LIN {X 0,Y 418.21,Z 141.387,A -85,B 0,C 180,E1 -10228.603,E2 -10228.603} C_VEL
LIN {X 0,Y 418.29,Z 141.379,A -85,B 0,C 180,E1 -10231.936,E2 -10231.936} C_VEL
LIN {X 0,Y 418.289,Z 141.382,A -85,B 0,C 180,E1 -10235.162,E2 -10235.162} C_VEL
LIN {X 0,Y 418.233,Z 141.384,A -85,B 0,C 180,E1 -10238.303,E2 -10238.303} C_VEL
LIN {X 0,Y 418.275,Z 141.384,A -85,B 0,C 180,E1 -10241.382,E2 -10241.382} C_VEL
LIN {X 0,Y 418.3,Z 141.376,A -85,B 0,C 180,E1 -10244.405,E2 -10244.405} C_VEL
LIN {X 0,Y 418.354,Z 141.373,A -85,B 0,C 180,E1 -10247.385,E2 -10247.385} C_VEL
LIN {X 0,Y 418.34,Z 141.371,A -85,B 0,C 180,E1 -10250.328,E2 -10250.328} C_VEL
LIN {X 0,Y 418.486,Z 141.357,A -85,B 0,C 180,E1 -10253.248,E2 -10253.248} C_VEL
LIN {X 0,Y 418.337,Z 141.375,A -85,B 0,C 180,E1 -10255.181,E2 -10255.181} C_VEL
LIN {X 0,Y 418.543,Z 141.346,A -85,B 0,C 180,E1 -10258.075,E2 -10258.075} C_VEL
LIN {X 0,Y 418.671,Z 141.33,A -85,B 0,C 180,E1 -10259.999,E2 -10259.999} C_VEL
LIN {X 0,Y 418.507,Z 141.356,A -85,B 0,C 180,E1 -10262.887,E2 -10262.887} C_VEL
LIN {X 0,Y 418.485,Z 141.36,A -85,B 0,C 180,E1 -10266.751,E2 -10266.751} C_VEL
LIN {X 0,Y 418.339,Z 141.371,A -85,B 0,C 180,E1 -10269.671,E2 -10269.671} C_VEL
LIN {X 0,Y 418.343,Z 141.373,A -85,B 0,C 180,E1 -10273,E2 -10273} C_VEL
LIN {X 0,Y 418.31,Z 141.379,A -85,B 0,C 180,E1 -10276.735,E2 -10276.735} C_VEL
LIN {X 0,Y 418.267,Z 141.381,A -85,B 0,C 180,E1 -10279.79,E2 -10279.79} C_VEL
LIN {X 0,Y 418.234,Z 141.387,A -85,B 0,C 180,E1 -10282.736,E2 -10282.736} C_VEL
LIN {X 0,Y 418.267,Z 141.382,A -85,B 0,C 180,E1 -10285.904,E2 -10285.904} C_VEL
LIN {X 0,Y 418.26,Z 141.381,A -85,B 0,C 180,E1 -10289.162,E2 -10289.162} C_VEL
LIN {X 0,Y 418.253,Z 141.382,A -85,B 0,C 180,E1 -10292.844,E2 -10292.844} C_VEL
LIN {X 0,Y 418.244,Z 141.388,A -85,B 0,C 180,E1 -10296.239,E2 -10296.239} C_VEL
LIN {X 0,Y 418.262,Z 141.384,A -85,B 0,C 180,E1 -10299.68,E2 -10299.68} C_VEL
LIN {X 0,Y 418.28,Z 141.381,A -85,B 0,C 180,E1 -10302.329,E2 -10302.329} C_VEL
LIN {X 0,Y 418.269,Z 141.38,A -85,B 0,C 180,E1 -10305.114,E2 -10305.114} C_VEL
LIN {X 0,Y 418.287,Z 141.383,A -85,B 0,C 180,E1 -10307.773,E2 -10307.773} C_VEL
LIN {X 0,Y 418.262,Z 141.385,A -85,B 0,C 180,E1 -10311.56,E2 -10311.56} C_VEL
LIN {X 0,Y 418.254,Z 141.383,A -85,B 0,C 180,E1 -10315.159,E2 -10315.159} C_VEL
LIN {X 0,Y 418.24,Z 141.388,A -85,B 0,C 180,E1 -10317.472,E2 -10317.472} C_VEL
LIN {X 0,Y 418.263,Z 141.381,A -85,B 0,C 180,E1 -10320.896,E2 -10320.896} C_VEL
LIN {X 0,Y 418.266,Z 141.381,A -85,B 0,C 180,E1 -10324.096,E2 -10324.096} C_VEL
LIN {X 0,Y 418.233,Z 141.389,A -85,B 0,C 180,E1 -10327.264,E2 -10327.264} C_VEL
LIN {X 0,Y 418.279,Z 141.378,A -85,B 0,C 180,E1 -10330.365,E2 -10330.365} C_VEL
LIN {X 0,Y 418.312,Z 141.381,A -85,B 0,C 180,E1 -10333.405,E2 -10333.405} C_VEL
LIN {X 0,Y 418.342,Z 141.374,A -85,B 0,C 180,E1 -10337,E2 -10337} C_VEL
LIN {X 0,Y 418.338,Z 141.371,A -85,B 0,C 180,E1 -10340.329,E2 -10340.329} C_VEL
LIN {X 0,Y 418.491,Z 141.358,A -85,B 0,C 180,E1 -10343.249,E2 -10343.249} C_VEL
LIN {X 0,Y 418.338,Z 141.377,A -85,B 0,C 180,E1 -10345.182,E2 -10345.182} C_VEL
LIN {X 0,Y 418.541,Z 141.346,A -85,B 0,C 180,E1 -10348.076,E2 -10348.076} C_VEL
LIN {X 0,Y 418.669,Z 141.33,A -85,B 0,C 180,E1 -10350.001,E2 -10350.001} C_VEL
LIN {X 0,Y 418.507,Z 141.357,A -85,B 0,C 180,E1 -10352.888,E2 -10352.888} C_VEL
LIN {X 0,Y 418.492,Z 141.358,A -85,B 0,C 180,E1 -10356.752,E2 -10356.752} C_VEL
LIN {X 0,Y 418.339,Z 141.371,A -85,B 0,C 180,E1 -10359.672,E2 -10359.672} C_VEL
LIN {X 0,Y 418.32,Z 141.377,A -85,B 0,C 180,E1 -10363.332,E2 -10363.332} C_VEL
LIN {X 0,Y 417.618,Z 141.465,A -85,B 0,C 180,E1 -10363.869,E2 -10363.869} C_VEL
LIN {X 0,Y 411.929,Z 142.175,A -85,B 0,C 180,E1 -10365.56,E2 -10365.56} C_VEL
LIN {X 0,Y 411.331,Z 142.25,A -85,B 0,C 180,E1 -10366.109,E2 -10366.109} C_VEL
LIN {X 0,Y 411.337,Z 142.3,A -85,B 0,C 180,E1 -10366.375,E2 -10366.375} C_VEL
LIN {X 0,Y 412.888,Z 151.501,A -85,B 0,C 180,E1 -10368.612,E2 -10368.612} C_VEL
LIN {X 0,Y 412.993,Z 152.785,A -85,B 0,C 180,E1 -10368.865,E2 -10368.865} C_VEL
LIN {X 0,Y 417.017,Z 172.236,A -85,B 0,C 180,E1 -10369.411,E2 -10369.411} C_VEL
LIN {X 0,Y 415.681,Z 260.265,A -85,B 0,C 180,E1 -10371.012,E2 -10371.012} C_VEL
LIN {X 0,Y 415.299,Z 273.928,A -85,B 0,C 180,E1 -10371.47,E2 -10371.47} C_VEL
LIN {X 0,Y 414.856,Z 286.236,A -85,B 0,C 180,E1 -10372.079,E2 -10372.079} C_VEL
LIN {X 0,Y 414.377,Z 297.489,A -85,B 0,C 180,E1 -10372.829,E2 -10372.829} C_VEL
LIN {X 0,Y 413.625,Z 308.356,A -85,B 0,C 180,E1 -10373.743,E2 -10373.743} C_VEL
LIN {X 0,Y 412.896,Z 319.455,A -85,B 0,C 180,E1 -10374.916,E2 -10374.916} C_VEL
LIN {X 0,Y 412.3,Z 328.343,A -85,B 0,C 180,E1 -10376.083,E2 -10376.083} C_VEL
LIN {X 0,Y 411.685,Z 336.809,A -85,B 0,C 180,E1 -10377.448,E2 -10377.448} C_VEL
LIN {X 0,Y 411.157,Z 344.341,A -85,B 0,C 180,E1 -10378.949,E2 -10378.949} C_VEL
LIN {X 0,Y 410.667,Z 350.919,A -85,B 0,C 180,E1 -10380.607,E2 -10380.607} C_VEL
LIN {X 0,Y 410.404,Z 355.393,A -85,B 0,C 180,E1 -10382.064,E2 -10382.064} C_VEL
LIN {X 0,Y 410.11,Z 359.41,A -85,B 0,C 180,E1 -10383.846,E2 -10383.846} C_VEL
LIN {X 0,Y 409.895,Z 362.062,A -85,B 0,C 180,E1 -10385.66,E2 -10385.66} C_VEL
LIN {X 0,Y 409.854,Z 363.037,A -85,B 0,C 180,E1 -10386.883,E2 -10386.883} C_VEL
LIN {X 0,Y 409.846,Z 363.428,A -85,B 0,C 180,E1 -10388.122,E2 -10388.122} C_VEL
LIN {X 0,Y 409.88,Z 363.07,A -85,B 0,C 180,E1 -10389.504,E2 -10389.504} C_VEL
LIN {X 0,Y 410.015,Z 361.754,A -85,B 0,C 180,E1 -10391.046,E2 -10391.046} C_VEL
LIN {X 0,Y 410.216,Z 359.494,A -85,B 0,C 180,E1 -10392.55,E2 -10392.55} C_VEL
LIN {X 0,Y 410.428,Z 356.324,A -85,B 0,C 180,E1 -10394.013,E2 -10394.013} C_VEL
LIN {X 0,Y 410.724,Z 352.199,A -85,B 0,C 180,E1 -10395.449,E2 -10395.449} C_VEL
LIN {X 0,Y 411.192,Z 347,A -85,B 0,C 180,E1 -10396.87,E2 -10396.87} C_VEL
LIN {X 0,Y 411.676,Z 340.719,A -85,B 0,C 180,E1 -10398.258,E2 -10398.258} C_VEL
LIN {X 0,Y 412.308,Z 333.087,A -85,B 0,C 180,E1 -10399.63,E2 -10399.63} C_VEL
LIN {X 0,Y 413.033,Z 323.793,A -85,B 0,C 180,E1 -10400.982,E2 -10400.982} C_VEL
LIN {X 0,Y 413.785,Z 313.743,A -85,B 0,C 180,E1 -10402.158,E2 -10402.158} C_VEL
LIN {X 0,Y 414.575,Z 303.217,A -85,B 0,C 180,E1 -10403.149,E2 -10403.149} C_VEL
LIN {X 0,Y 415.31,Z 291.58,A -85,B 0,C 180,E1 -10404.015,E2 -10404.015} C_VEL
LIN {X 0,Y 415.854,Z 279.546,A -85,B 0,C 180,E1 -10404.694,E2 -10404.694} C_VEL
LIN {X 0,Y 416.243,Z 267.043,A -85,B 0,C 180,E1 -10405.202,E2 -10405.202} C_VEL
LIN {X 0,Y 416.569,Z 254.522,A -85,B 0,C 180,E1 -10405.52,E2 -10405.52} C_VEL
LIN {X 0,Y 417.79,Z 172.296,A -85,B 0,C 180,E1 -10407.018,E2 -10407.018} C_VEL
LIN {X 0,Y 413.907,Z 155.246,A -85,B 0,C 180,E1 -10407.558,E2 -10407.558} C_VEL
LIN {X 0,Y 413.389,Z 153.267,A -85,B 0,C 180,E1 -10407.657,E2 -10407.657} C_VEL
LIN {X 0,Y 411.253,Z 142.258,A -85,B 0,C 180,E1 -10410.349,E2 -10410.349} C_VEL
LIN {X 0,Y 411.236,Z 142.264,A -85,B 0,C 180,E1 -10413.62,E2 -10413.62} C_VEL
LIN {X 0,Y 411.198,Z 142.27,A -85,B 0,C 180,E1 -10416.853,E2 -10416.853} C_VEL
LIN {X 0,Y 411.218,Z 142.262,A -85,B 0,C 180,E1 -10420.051,E2 -10420.051} C_VEL
LIN {X 0,Y 411.267,Z 142.259,A -85,B 0,C 180,E1 -10423.132,E2 -10423.132} C_VEL
LIN {X 0,Y 411.31,Z 142.253,A -85,B 0,C 180,E1 -10426.897,E2 -10426.897} C_VEL
LIN {X 0,Y 411.294,Z 142.252,A -85,B 0,C 180,E1 -10430.162,E2 -10430.162} C_VEL
LIN {X 0,Y 411.395,Z 142.24,A -85,B 0,C 180,E1 -10433.133,E2 -10433.133} C_VEL
LIN {X 0,Y 411.295,Z 142.25,A -85,B 0,C 180,E1 -10435.099,E2 -10435.099} C_VEL
LIN {X 0,Y 411.507,Z 142.229,A -85,B 0,C 180,E1 -10438.043,E2 -10438.043} C_VEL
LIN {X 0,Y 411.385,Z 142.239,A -85,B 0,C 180,E1 -10440.979,E2 -10440.979} C_VEL
LIN {X 0,Y 411.431,Z 142.227,A -85,B 0,C 180,E1 -10442.938,E2 -10442.938} C_VEL
LIN {X 0,Y 411.432,Z 142.235,A -85,B 0,C 180,E1 -10445.883,E2 -10445.883} C_VEL
LIN {X 0,Y 411.31,Z 142.247,A -85,B 0,C 180,E1 -10448.847,E2 -10448.847} C_VEL
LIN {X 0,Y 411.273,Z 142.251,A -85,B 0,C 180,E1 -10451.834,E2 -10451.834} C_VEL
LIN {X 0,Y 411.211,Z 142.255,A -85,B 0,C 180,E1 -10454.855,E2 -10454.855} C_VEL
LIN {X 0,Y 411.161,Z 142.267,A -85,B 0,C 180,E1 -10457.92,E2 -10457.92} C_VEL
LIN {X 0,Y 411.182,Z 142.264,A -85,B 0,C 180,E1 -10461.035,E2 -10461.035} C_VEL
LIN {X 0,Y 411.176,Z 142.262,A -85,B 0,C 180,E1 -10464.219,E2 -10464.219} C_VEL
LIN {X 0,Y 411.145,Z 142.266,A -85,B 0,C 180,E1 -10467.486,E2 -10467.486} C_VEL
LIN {X 0,Y 411.197,Z 142.263,A -85,B 0,C 180,E1 -10469.714,E2 -10469.714} C_VEL
LIN {X 0,Y 411.209,Z 142.266,A -85,B 0,C 180,E1 -10473.156,E2 -10473.156} C_VEL
LIN {X 0,Y 411.197,Z 142.264,A -85,B 0,C 180,E1 -10476.552,E2 -10476.552} C_VEL
LIN {X 0,Y 411.174,Z 142.266,A -85,B 0,C 180,E1 -10479.72,E2 -10479.72} C_VEL
LIN {X 0,Y 411.167,Z 142.268,A -85,B 0,C 180,E1 -10483.135,E2 -10483.135} C_VEL
LIN {X 0,Y 411.17,Z 142.269,A -85,B 0,C 180,E1 -10485.881,E2 -10485.881} C_VEL
LIN {X 0,Y 411.156,Z 142.272,A -85,B 0,C 180,E1 -10488.774,E2 -10488.774} C_VEL
LIN {X 0,Y 411.191,Z 142.268,A -85,B 0,C 180,E1 -10492.025,E2 -10492.025} C_VEL
LIN {X 0,Y 411.211,Z 142.264,A -85,B 0,C 180,E1 -10495.666,E2 -10495.666} C_VEL
LIN {X 0,Y 411.194,Z 142.267,A -85,B 0,C 180,E1 -10499.152,E2 -10499.152} C_VEL
LIN {X 0,Y 411.26,Z 142.396,A -85,B 0,C 180,E1 -10501.489,E2 -10501.489} C_VEL
LIN {X 0,Y 413.905,Z 154.634,A -85,B 0,C 180,E1 -10504.149,E2 -10504.149} C_VEL
LIN {X 0,Y 414.568,Z 159.685,A -85,B 0,C 180,E1 -10505.191,E2 -10505.191} C_VEL
LIN {X 0,Y 413.326,Z 177.24,A -85,B 0,C 180,E1 -10508.556,E2 -10508.556} C_VEL
LIN {X 0,Y 412.781,Z 186.857,A -85,B 0,C 180,E1 -10510.376,E2 -10510.376} C_VEL
LIN {X 0,Y 416.686,Z 211.598,A -85,B 0,C 180,E1 -10511.057,E2 -10511.057} C_VEL
LIN {X 0,Y 417.247,Z 218.282,A -85,B 0,C 180,E1 -10511.212,E2 -10511.212} C_VEL
LIN {X 0,Y 416.163,Z 296.183,A -85,B 0,C 180,E1 -10512.652,E2 -10512.652} C_VEL
LIN {X 0,Y 415.507,Z 309.921,A -85,B 0,C 180,E1 -10513.099,E2 -10513.099} C_VEL
LIN {X 0,Y 414.819,Z 322.351,A -85,B 0,C 180,E1 -10513.703,E2 -10513.703} C_VEL
LIN {X 0,Y 414.049,Z 334.29,A -85,B 0,C 180,E1 -10514.493,E2 -10514.493} C_VEL
LIN {X 0,Y 413.192,Z 346.036,A -85,B 0,C 180,E1 -10515.495,E2 -10515.495} C_VEL
LIN {X 0,Y 412.425,Z 356.164,A -85,B 0,C 180,E1 -10516.574,E2 -10516.574} C_VEL
LIN {X 0,Y 411.663,Z 366.341,A -85,B 0,C 180,E1 -10517.928,E2 -10517.928} C_VEL
LIN {X 0,Y 410.915,Z 375.306,A -85,B 0,C 180,E1 -10519.405,E2 -10519.405} C_VEL
LIN {X 0,Y 410.462,Z 382.511,A -85,B 0,C 180,E1 -10520.887,E2 -10520.887} C_VEL
LIN {X 0,Y 410.174,Z 389.097,A -85,B 0,C 180,E1 -10522.616,E2 -10522.616} C_VEL
LIN {X 0,Y 409.99,Z 393.452,A -85,B 0,C 180,E1 -10524.096,E2 -10524.096} C_VEL
LIN {X 0,Y 410.009,Z 395.771,A -85,B 0,C 180,E1 -10525.083,E2 -10525.083} C_VEL
LIN {X 0,Y 409.941,Z 397.615,A -85,B 0,C 180,E1 -10526.067,E2 -10526.067} C_VEL
LIN {X 0,Y 409.973,Z 399.015,A -85,B 0,C 180,E1 -10527.052,E2 -10527.052} C_VEL
LIN {X 0,Y 410.02,Z 400.015,A -85,B 0,C 180,E1 -10528.035,E2 -10528.035} C_VEL
LIN {X 0,Y 409.983,Z 400.617,A -85,B 0,C 180,E1 -10529.017,E2 -10529.017} C_VEL
LIN {X 0,Y 409.979,Z 400.785,A -85,B 0,C 180,E1 -10529.999,E2 -10529.999} C_VEL
LIN {X 0,Y 409.983,Z 400.538,A -85,B 0,C 180,E1 -10530.982,E2 -10530.982} C_VEL
LIN {X 0,Y 410.02,Z 399.899,A -85,B 0,C 180,E1 -10531.964,E2 -10531.964} C_VEL
LIN {X 0,Y 409.976,Z 398.86,A -85,B 0,C 180,E1 -10532.947,E2 -10532.947} C_VEL
LIN {X 0,Y 409.943,Z 397.366,A -85,B 0,C 180,E1 -10533.932,E2 -10533.932} C_VEL
LIN {X 0,Y 410.002,Z 394.315,A -85,B 0,C 180,E1 -10535.409,E2 -10535.409} C_VEL
LIN {X 0,Y 410.095,Z 390.185,A -85,B 0,C 180,E1 -10536.889,E2 -10536.889} C_VEL
LIN {X 0,Y 410.373,Z 383.845,A -85,B 0,C 180,E1 -10538.618,E2 -10538.618} C_VEL
LIN {X 0,Y 410.733,Z 376.931,A -85,B 0,C 180,E1 -10540.101,E2 -10540.101} C_VEL
LIN {X 0,Y 411.244,Z 369.875,A -85,B 0,C 180,E1 -10541.334,E2 -10541.334} C_VEL
LIN {X 0,Y 411.812,Z 361.367,A -85,B 0,C 180,E1 -10542.567,E2 -10542.567} C_VEL
LIN {X 0,Y 412.504,Z 350.848,A -85,B 0,C 180,E1 -10543.799,E2 -10543.799} C_VEL
LIN {X 0,Y 413.334,Z 339.017,A -85,B 0,C 180,E1 -10544.902,E2 -10544.902} C_VEL
LIN {X 0,Y 414.107,Z 327.155,A -85,B 0,C 180,E1 -10545.756,E2 -10545.756} C_VEL
LIN {X 0,Y 414.793,Z 314.852,A -85,B 0,C 180,E1 -10546.423,E2 -10546.423} C_VEL
LIN {X 0,Y 415.336,Z 302.328,A -85,B 0,C 180,E1 -10546.907,E2 -10546.907} C_VEL
LIN {X 0,Y 415.652,Z 287.89,A -85,B 0,C 180,E1 -10547.242,E2 -10547.242} C_VEL
LIN {X 0,Y 416.483,Z 215.312,A -85,B 0,C 180,E1 -10548.55,E2 -10548.55} C_VEL
LIN {X 0,Y 412.522,Z 188.027,A -85,B 0,C 180,E1 -10549.241,E2 -10549.241} C_VEL
LIN {X 0,Y 413.776,Z 168.398,A -85,B 0,C 180,E1 -10552.995,E2 -10552.995} C_VEL
LIN {X 0,Y 414.447,Z 158.976,A -85,B 0,C 180,E1 -10554.815,E2 -10554.815} C_VEL
LIN {X 0,Y 413.035,Z 150.76,A -85,B 0,C 180,E1 -10556.529,E2 -10556.529} C_VEL
LIN {X 0,Y 411.316,Z 142.251,A -85,B 0,C 180,E1 -10558.373,E2 -10558.373} C_VEL
LIN {X 0,Y 411.167,Z 142.271,A -85,B 0,C 180,E1 -10561.997,E2 -10561.997} C_VEL
LIN {X 0,Y 411.211,Z 142.259,A -85,B 0,C 180,E1 -10564.878,E2 -10564.878} C_VEL
LIN {X 0,Y 411.208,Z 142.263,A -85,B 0,C 180,E1 -10568.168,E2 -10568.168} C_VEL
LIN {X 0,Y 411.165,Z 142.266,A -85,B 0,C 180,E1 -10571.228,E2 -10571.228} C_VEL
LIN {X 0,Y 411.176,Z 142.264,A -85,B 0,C 180,E1 -10574.49,E2 -10574.49} C_VEL
LIN {X 0,Y 411.177,Z 142.265,A -85,B 0,C 180,E1 -10578.194,E2 -10578.194} C_VEL
LIN {X 0,Y 411.21,Z 142.259,A -85,B 0,C 180,E1 -10580.774,E2 -10580.774} C_VEL
LIN {X 0,Y 411.196,Z 142.261,A -85,B 0,C 180,E1 -10584.471,E2 -10584.471} C_VEL
LIN {X 0,Y 411.206,Z 142.26,A -85,B 0,C 180,E1 -10586.873,E2 -10586.873} C_VEL
LIN {X 0,Y 411.232,Z 142.256,A -85,B 0,C 180,E1 -10590.644,E2 -10590.644} C_VEL
LIN {X 0,Y 411.237,Z 142.26,A -85,B 0,C 180,E1 -10593.619,E2 -10593.619} C_VEL
LIN {X 0,Y 411.202,Z 142.262,A -85,B 0,C 180,E1 -10596.852,E2 -10596.852} C_VEL
LIN {X 0,Y 411.213,Z 142.259,A -85,B 0,C 180,E1 -10600.05,E2 -10600.05} C_VEL
LIN {X 0,Y 411.261,Z 142.259,A -85,B 0,C 180,E1 -10603.131,E2 -10603.131} C_VEL
LIN {X 0,Y 411.304,Z 142.252,A -85,B 0,C 180,E1 -10606.895,E2 -10606.895} C_VEL
LIN {X 0,Y 411.292,Z 142.249,A -85,B 0,C 180,E1 -10610.161,E2 -10610.161} C_VEL
LIN {X 0,Y 411.45,Z 142.234,A -85,B 0,C 180,E1 -10613.132,E2 -10613.132} C_VEL
LIN {X 0,Y 411.308,Z 142.252,A -85,B 0,C 180,E1 -10615.098,E2 -10615.098} C_VEL
LIN {X 0,Y 411.512,Z 142.221,A -85,B 0,C 180,E1 -10618.042,E2 -10618.042} C_VEL
LIN {X 0,Y 411.64,Z 142.205,A -85,B 0,C 180,E1 -10619.999,E2 -10619.999} C_VEL
LIN {X 0,Y 411.463,Z 142.233,A -85,B 0,C 180,E1 -10622.937,E2 -10622.937} C_VEL
LIN {X 0,Y 411.449,Z 142.234,A -85,B 0,C 180,E1 -10626.867,E2 -10626.867} C_VEL
LIN {X 0,Y 411.291,Z 142.249,A -85,B 0,C 180,E1 -10629.838,E2 -10629.838} C_VEL
LIN {X 0,Y 411.302,Z 142.249,A -85,B 0,C 180,E1 -10633.104,E2 -10633.104} C_VEL
LIN {X 0,Y 411.259,Z 142.256,A -85,B 0,C 180,E1 -10636.868,E2 -10636.868} C_VEL
LIN {X 0,Y 411.227,Z 142.259,A -85,B 0,C 180,E1 -10639.986,E2 -10639.986} C_VEL
LIN {X 0,Y 411.199,Z 142.261,A -85,B 0,C 180,E1 -10643.147,E2 -10643.147} C_VEL
LIN {X 0,Y 411.234,Z 142.262,A -85,B 0,C 180,E1 -10646.38,E2 -10646.38} C_VEL
LIN {X 0,Y 411.196,Z 142.262,A -85,B 0,C 180,E1 -10649.712,E2 -10649.712} C_VEL
LIN {X 0,Y 411.202,Z 142.26,A -85,B 0,C 180,E1 -10653.155,E2 -10653.155} C_VEL
LIN {X 0,Y 411.191,Z 142.263,A -85,B 0,C 180,E1 -10656.553,E2 -10656.553} C_VEL
LIN {X 0,Y 411.224,Z 142.261,A -85,B 0,C 180,E1 -10659.73,E2 -10659.73} C_VEL
LIN {X 0,Y 411.226,Z 142.257,A -85,B 0,C 180,E1 -10663.126,E2 -10663.126} C_VEL
LIN {X 0,Y 411.235,Z 142.263,A -85,B 0,C 180,E1 -10665.871,E2 -10665.871} C_VEL
LIN {X 0,Y 411.205,Z 142.26,A -85,B 0,C 180,E1 -10668.764,E2 -10668.764} C_VEL
LIN {X 0,Y 411.2,Z 142.264,A -85,B 0,C 180,E1 -10672.028,E2 -10672.028} C_VEL
LIN {X 0,Y 411.201,Z 142.267,A -85,B 0,C 180,E1 -10675.667,E2 -10675.667} C_VEL
LIN {X 0,Y 411.184,Z 142.264,A -85,B 0,C 180,E1 -10679.153,E2 -10679.153} C_VEL
LIN {X 0,Y 411.254,Z 142.253,A -85,B 0,C 180,E1 -10682.523,E2 -10682.523} C_VEL
LIN {X 0,Y 411.222,Z 142.261,A -85,B 0,C 180,E1 -10685.785,E2 -10685.785} C_VEL
LIN {X 0,Y 411.192,Z 142.263,A -85,B 0,C 180,E1 -10688.966,E2 -10688.966} C_VEL
LIN {X 0,Y 411.248,Z 142.255,A -85,B 0,C 180,E1 -10692.085,E2 -10692.085} C_VEL
LIN {X 0,Y 411.256,Z 142.258,A -85,B 0,C 180,E1 -10695.148,E2 -10695.148} C_VEL
LIN {X 0,Y 411.28,Z 142.25,A -85,B 0,C 180,E1 -10698.168,E2 -10698.168} C_VEL
LIN {X 0,Y 411.478,Z 142.225,A -85,B 0,C 180,E1 -10702.147,E2 -10702.147} C_VEL
LIN {X 0,Y 411.473,Z 142.226,A -85,B 0,C 180,E1 -10704.119,E2 -10704.119} C_VEL
LIN {X 0,Y 411.51,Z 142.221,A -85,B 0,C 180,E1 -10708.043,E2 -10708.043} C_VEL
LIN {X 0,Y 411.639,Z 142.205,A -85,B 0,C 180,E1 -10710.001,E2 -10710.001} C_VEL
LIN {X 0,Y 411.463,Z 142.235,A -85,B 0,C 180,E1 -10712.938,E2 -10712.938} C_VEL
LIN {X 0,Y 411.458,Z 142.235,A -85,B 0,C 180,E1 -10716.868,E2 -10716.868} C_VEL
LIN {X 0,Y 411.291,Z 142.249,A -85,B 0,C 180,E1 -10719.839,E2 -10719.839} C_VEL
LIN {X 0,Y 411.284,Z 142.253,A -85,B 0,C 180,E1 -10723.32,E2 -10723.32} C_VEL
LIN {X 0,Y 411.331,Z 142.25,A -85,B 0,C 180,E1 -10726.109,E2 -10726.109} C_VEL
LIN {X 0,Y 411.267,Z 142.94,A -85,B 0,C 180,E1 -10726.499,E2 -10726.499} C_VEL
LIN {X 0,Y 410.694,Z 145.504,A -85,B 0,C 180,E1 -10727.091,E2 -10727.091} C_VEL
LIN {X 0,Y 409.217,Z 149.691,A -85,B 0,C 180,E1 -10727.933,E2 -10727.933} C_VEL
LIN {X 0,Y 408.351,Z 154.177,A -85,B 0,C 180,E1 -10728.364,E2 -10728.364} C_VEL
LIN {X 0,Y 407.985,Z 159.599,A -85,B 0,C 180,E1 -10728.712,E2 -10728.712} C_VEL
LIN {X 0,Y 408.345,Z 163.41,A -85,B 0,C 180,E1 -10728.858,E2 -10728.858} C_VEL
LIN {X 0,Y 410.228,Z 173.002,A -85,B 0,C 180,E1 -10729.125,E2 -10729.125} C_VEL
LIN {X 0,Y 408.875,Z 259.99,A -85,B 0,C 180,E1 -10730.731,E2 -10730.731} C_VEL
LIN {X 0,Y 408.466,Z 273.511,A -85,B 0,C 180,E1 -10731.182,E2 -10731.182} C_VEL
LIN {X 0,Y 408.031,Z 285.861,A -85,B 0,C 180,E1 -10731.793,E2 -10731.793} C_VEL
LIN {X 0,Y 407.518,Z 297.436,A -85,B 0,C 180,E1 -10732.565,E2 -10732.565} C_VEL
LIN {X 0,Y 406.701,Z 308.993,A -85,B 0,C 180,E1 -10733.553,E2 -10733.553} C_VEL
LIN {X 0,Y 405.986,Z 319.521,A -85,B 0,C 180,E1 -10734.685,E2 -10734.685} C_VEL
LIN {X 0,Y 405.298,Z 329.093,A -85,B 0,C 180,E1 -10735.967,E2 -10735.967} C_VEL
LIN {X 0,Y 404.63,Z 337.874,A -85,B 0,C 180,E1 -10737.425,E2 -10737.425} C_VEL
LIN {X 0,Y 404.131,Z 344.84,A -85,B 0,C 180,E1 -10738.855,E2 -10738.855} C_VEL
LIN {X 0,Y 403.678,Z 350.622,A -85,B 0,C 180,E1 -10740.325,E2 -10740.325} C_VEL
LIN {X 0,Y 403.301,Z 356.025,A -85,B 0,C 180,E1 -10742.107,E2 -10742.107} C_VEL
LIN {X 0,Y 403.026,Z 359.958,A -85,B 0,C 180,E1 -10743.92,E2 -10743.92} C_VEL
LIN {X 0,Y 402.853,Z 361.822,A -85,B 0,C 180,E1 -10745.15,E2 -10745.15} C_VEL
LIN {X 0,Y 402.769,Z 363.225,A -85,B 0,C 180,E1 -10746.616,E2 -10746.616} C_VEL
LIN {X 0,Y 402.765,Z 363.752,A -85,B 0,C 180,E1 -10748.26,E2 -10748.26} C_VEL
LIN {X 0,Y 402.823,Z 362.965,A -85,B 0,C 180,E1 -10750.207,E2 -10750.207} C_VEL
LIN {X 0,Y 403.078,Z 360.668,A -85,B 0,C 180,E1 -10752.167,E2 -10752.167} C_VEL
LIN {X 0,Y 403.275,Z 358.103,A -85,B 0,C 180,E1 -10753.52,E2 -10753.52} C_VEL
LIN {X 0,Y 403.548,Z 354.525,A -85,B 0,C 180,E1 -10754.942,E2 -10754.942} C_VEL
LIN {X 0,Y 404.033,Z 348.955,A -85,B 0,C 180,E1 -10756.638,E2 -10756.638} C_VEL
LIN {X 0,Y 404.651,Z 341.748,A -85,B 0,C 180,E1 -10758.317,E2 -10758.317} C_VEL
LIN {X 0,Y 405.322,Z 334.19,A -85,B 0,C 180,E1 -10759.724,E2 -10759.724} C_VEL
LIN {X 0,Y 406.102,Z 324.741,A -85,B 0,C 180,E1 -10761.149,E2 -10761.149} C_VEL
LIN {X 0,Y 406.911,Z 314.507,A -85,B 0,C 180,E1 -10762.378,E2 -10762.378} C_VEL
LIN {X 0,Y 407.841,Z 302.963,A -85,B 0,C 180,E1 -10763.481,E2 -10763.481} C_VEL
LIN {X 0,Y 408.525,Z 292.263,A -85,B 0,C 180,E1 -10764.287,E2 -10764.287} C_VEL
LIN {X 0,Y 409.116,Z 279.829,A -85,B 0,C 180,E1 -10765.002,E2 -10765.002} C_VEL
LIN {X 0,Y 409.587,Z 266.535,A -85,B 0,C 180,E1 -10765.543,E2 -10765.543} C_VEL
LIN {X 0,Y 409.9,Z 252.754,A -85,B 0,C 180,E1 -10765.877,E2 -10765.877} C_VEL
LIN {X 0,Y 411.101,Z 173.169,A -85,B 0,C 180,E1 -10767.36,E2 -10767.36} C_VEL
LIN {X 0,Y 407.478,Z 157.271,A -85,B 0,C 180,E1 -10767.878,E2 -10767.878} C_VEL
LIN {X 0,Y 406.336,Z 153.66,A -85,B 0,C 180,E1 -10768.043,E2 -10768.043} C_VEL
LIN {X 0,Y 404.21,Z 143.137,A -85,B 0,C 180,E1 -10770.675,E2 -10770.675} C_VEL
LIN {X 0,Y 404.196,Z 143.141,A -85,B 0,C 180,E1 -10773.124,E2 -10773.124} C_VEL
LIN {X 0,Y 404.173,Z 143.147,A -85,B 0,C 180,E1 -10775.335,E2 -10775.335} C_VEL
LIN {X 0,Y 404.141,Z 143.147,A -85,B 0,C 180,E1 -10778.581,E2 -10778.581} C_VEL
LIN {X 0,Y 404.208,Z 143.134,A -85,B 0,C 180,E1 -10781.762,E2 -10781.762} C_VEL
LIN {X 0,Y 404.209,Z 143.137,A -85,B 0,C 180,E1 -10784.883,E2 -10784.883} C_VEL
LIN {X 0,Y 404.26,Z 143.13,A -85,B 0,C 180,E1 -10787.959,E2 -10787.959} C_VEL
LIN {X 0,Y 404.27,Z 143.131,A -85,B 0,C 180,E1 -10790.999,E2 -10790.999} C_VEL
LIN {X 0,Y 404.382,Z 143.115,A -85,B 0,C 180,E1 -10794.015,E2 -10794.015} C_VEL
LIN {X 0,Y 404.476,Z 143.104,A -85,B 0,C 180,E1 -10798.009,E2 -10798.009} C_VEL
LIN {X 0,Y 404.355,Z 143.115,A -85,B 0,C 180,E1 -10800.996,E2 -10800.996} C_VEL
LIN {X 0,Y 404.364,Z 143.107,A -85,B 0,C 180,E1 -10802.989,E2 -10802.989} C_VEL
LIN {X 0,Y 404.381,Z 143.111,A -85,B 0,C 180,E1 -10805.986,E2 -10805.986} C_VEL
LIN {X 0,Y 404.259,Z 143.126,A -85,B 0,C 180,E1 -10809.002,E2 -10809.002} C_VEL
LIN {X 0,Y 404.248,Z 143.128,A -85,B 0,C 180,E1 -10812.042,E2 -10812.042} C_VEL
LIN {X 0,Y 404.16,Z 143.134,A -85,B 0,C 180,E1 -10815.12,E2 -10815.12} C_VEL
LIN {X 0,Y 404.122,Z 143.141,A -85,B 0,C 180,E1 -10818.243,E2 -10818.243} C_VEL
LIN {X 0,Y 404.129,Z 143.147,A -85,B 0,C 180,E1 -10821.42,E2 -10821.42} C_VEL
LIN {X 0,Y 404.132,Z 143.14,A -85,B 0,C 180,E1 -10824.669,E2 -10824.669} C_VEL
LIN {X 0,Y 404.104,Z 143.142,A -85,B 0,C 180,E1 -10828.007,E2 -10828.007} C_VEL
LIN {X 0,Y 404.144,Z 143.141,A -85,B 0,C 180,E1 -10830.286,E2 -10830.286} C_VEL
LIN {X 0,Y 404.143,Z 143.141,A -85,B 0,C 180,E1 -10833.813,E2 -10833.813} C_VEL
LIN {X 0,Y 404.14,Z 143.147,A -85,B 0,C 180,E1 -10836.874,E2 -10836.874} C_VEL
LIN {X 0,Y 404.122,Z 143.145,A -85,B 0,C 180,E1 -10840.075,E2 -10840.075} C_VEL
LIN {X 0,Y 404.147,Z 143.143,A -85,B 0,C 180,E1 -10843.082,E2 -10843.082} C_VEL
LIN {X 0,Y 404.151,Z 143.144,A -85,B 0,C 180,E1 -10845.926,E2 -10845.926} C_VEL
LIN {X 0,Y 404.111,Z 143.15,A -85,B 0,C 180,E1 -10848.633,E2 -10848.633} C_VEL
LIN {X 0,Y 404.146,Z 143.143,A -85,B 0,C 180,E1 -10851.494,E2 -10851.494} C_VEL
LIN {X 0,Y 404.189,Z 143.137,A -85,B 0,C 180,E1 -10854.984,E2 -10854.984} C_VEL
LIN {X 0,Y 404.147,Z 143.148,A -85,B 0,C 180,E1 -10858.554,E2 -10858.554} C_VEL
LIN {X 0,Y 404.221,Z 143.248,A -85,B 0,C 180,E1 -10861.152,E2 -10861.152} C_VEL
LIN {X 0,Y 407.079,Z 156.52,A -85,B 0,C 180,E1 -10864.097,E2 -10864.097} C_VEL
LIN {X 0,Y 407.663,Z 160.87,A -85,B 0,C 180,E1 -10865.015,E2 -10865.015} C_VEL
LIN {X 0,Y 406.459,Z 177.079,A -85,B 0,C 180,E1 -10868.176,E2 -10868.176} C_VEL
LIN {X 0,Y 405.905,Z 186.428,A -85,B 0,C 180,E1 -10869.987,E2 -10869.987} C_VEL
LIN {X 0,Y 409.976,Z 211.997,A -85,B 0,C 180,E1 -10870.719,E2 -10870.719} C_VEL
LIN {X 0,Y 410.59,Z 218.448,A -85,B 0,C 180,E1 -10870.878,E2 -10870.878} C_VEL
LIN {X 0,Y 409.447,Z 295.555,A -85,B 0,C 180,E1 -10872.325,E2 -10872.325} C_VEL
LIN {X 0,Y 408.786,Z 309.375,A -85,B 0,C 180,E1 -10872.78,E2 -10872.78} C_VEL
LIN {X 0,Y 408.081,Z 321.3,A -85,B 0,C 180,E1 -10873.362,E2 -10873.362} C_VEL
LIN {X 0,Y 407.35,Z 332.643,A -85,B 0,C 180,E1 -10874.103,E2 -10874.103} C_VEL
LIN {X 0,Y 406.39,Z 344.373,A -85,B 0,C 180,E1 -10875.093,E2 -10875.093} C_VEL
LIN {X 0,Y 405.523,Z 355.952,A -85,B 0,C 180,E1 -10876.333,E2 -10876.333} C_VEL
LIN {X 0,Y 404.854,Z 364.496,A -85,B 0,C 180,E1 -10877.467,E2 -10877.467} C_VEL
LIN {X 0,Y 403.998,Z 373.707,A -85,B 0,C 180,E1 -10878.967,E2 -10878.967} C_VEL
LIN {X 0,Y 403.536,Z 381.152,A -85,B 0,C 180,E1 -10880.476,E2 -10880.476} C_VEL
LIN {X 0,Y 403.192,Z 387.135,A -85,B 0,C 180,E1 -10881.984,E2 -10881.984} C_VEL
LIN {X 0,Y 402.934,Z 392.751,A -85,B 0,C 180,E1 -10883.828,E2 -10883.828} C_VEL
LIN {X 0,Y 402.917,Z 395.48,A -85,B 0,C 180,E1 -10884.996,E2 -10884.996} C_VEL
LIN {X 0,Y 402.859,Z 397.314,A -85,B 0,C 180,E1 -10885.998,E2 -10885.998} C_VEL
LIN {X 0,Y 402.948,Z 399.705,A -85,B 0,C 180,E1 -10888,E2 -10888} C_VEL
LIN {X 0,Y 402.908,Z 400.3,A -85,B 0,C 180,E1 -10889,E2 -10889} C_VEL
LIN {X 0,Y 402.901,Z 400.457,A -85,B 0,C 180,E1 -10889.999,E2 -10889.999} C_VEL
LIN {X 0,Y 402.907,Z 400.204,A -85,B 0,C 180,E1 -10890.999,E2 -10890.999} C_VEL
LIN {X 0,Y 402.948,Z 399.559,A -85,B 0,C 180,E1 -10891.998,E2 -10891.998} C_VEL
LIN {X 0,Y 402.876,Z 398.51,A -85,B 0,C 180,E1 -10892.999,E2 -10892.999} C_VEL
LIN {X 0,Y 402.863,Z 397.002,A -85,B 0,C 180,E1 -10894.001,E2 -10894.001} C_VEL
LIN {X 0,Y 402.9,Z 393.932,A -85,B 0,C 180,E1 -10895.505,E2 -10895.505} C_VEL
LIN {X 0,Y 403.038,Z 389.785,A -85,B 0,C 180,E1 -10897.011,E2 -10897.011} C_VEL
LIN {X 0,Y 403.323,Z 383.422,A -85,B 0,C 180,E1 -10898.77,E2 -10898.77} C_VEL
LIN {X 0,Y 403.687,Z 376.483,A -85,B 0,C 180,E1 -10900.279,E2 -10900.279} C_VEL
LIN {X 0,Y 404.344,Z 367.804,A -85,B 0,C 180,E1 -10901.784,E2 -10901.784} C_VEL
LIN {X 0,Y 404.977,Z 358.886,A -85,B 0,C 180,E1 -10903.038,E2 -10903.038} C_VEL
LIN {X 0,Y 405.695,Z 349.099,A -85,B 0,C 180,E1 -10904.163,E2 -10904.163} C_VEL
LIN {X 0,Y 406.43,Z 338.388,A -85,B 0,C 180,E1 -10905.161,E2 -10905.161} C_VEL
LIN {X 0,Y 407.233,Z 326.411,A -85,B 0,C 180,E1 -10906.029,E2 -10906.029} C_VEL
LIN {X 0,Y 407.913,Z 313.979,A -85,B 0,C 180,E1 -10906.708,E2 -10906.708} C_VEL
LIN {X 0,Y 408.531,Z 301.206,A -85,B 0,C 180,E1 -10907.198,E2 -10907.198} C_VEL
LIN {X 0,Y 408.895,Z 286.145,A -85,B 0,C 180,E1 -10907.537,E2 -10907.537} C_VEL
LIN {X 0,Y 409.7,Z 216.271,A -85,B 0,C 180,E1 -10908.82,E2 -10908.82} C_VEL
LIN {X 0,Y 405.572,Z 187.749,A -85,B 0,C 180,E1 -10909.551,E2 -10909.551} C_VEL
LIN {X 0,Y 406.942,Z 167.95,A -85,B 0,C 180,E1 -10913.404,E2 -10913.404} C_VEL
LIN {X 0,Y 407.469,Z 159.879,A -85,B 0,C 180,E1 -10914.997,E2 -10914.997} C_VEL
LIN {X 0,Y 405.481,Z 148.999,A -85,B 0,C 180,E1 -10917.319,E2 -10917.319} C_VEL
LIN {X 0,Y 404.244,Z 143.133,A -85,B 0,C 180,E1 -10918.632,E2 -10918.632} C_VEL
LIN {X 0,Y 404.142,Z 143.144,A -85,B 0,C 180,E1 -10922.621,E2 -10922.621} C_VEL
LIN {X 0,Y 404.182,Z 143.135,A -85,B 0,C 180,E1 -10925.189,E2 -10925.189} C_VEL
LIN {X 0,Y 404.158,Z 143.138,A -85,B 0,C 180,E1 -10928.756,E2 -10928.756} C_VEL
LIN {X 0,Y 404.124,Z 143.146,A -85,B 0,C 180,E1 -10931.599,E2 -10931.599} C_VEL
LIN {X 0,Y 404.145,Z 143.139,A -85,B 0,C 180,E1 -10934.521,E2 -10934.521} C_VEL
LIN {X 0,Y 404.136,Z 143.143,A -85,B 0,C 180,E1 -10937.295,E2 -10937.295} C_VEL
LIN {X 0,Y 404.168,Z 143.14,A -85,B 0,C 180,E1 -10939.955,E2 -10939.955} C_VEL
LIN {X 0,Y 404.135,Z 143.142,A -85,B 0,C 180,E1 -10943.125,E2 -10943.125} C_VEL
LIN {X 0,Y 404.144,Z 143.14,A -85,B 0,C 180,E1 -10946.187,E2 -10946.187} C_VEL
LIN {X 0,Y 404.144,Z 143.143,A -85,B 0,C 180,E1 -10949.714,E2 -10949.714} C_VEL
LIN {X 0,Y 404.195,Z 143.137,A -85,B 0,C 180,E1 -10953.122,E2 -10953.122} C_VEL
LIN {X 0,Y 404.177,Z 143.142,A -85,B 0,C 180,E1 -10955.334,E2 -10955.334} C_VEL
LIN {X 0,Y 404.137,Z 143.141,A -85,B 0,C 180,E1 -10958.58,E2 -10958.58} C_VEL
LIN {X 0,Y 404.203,Z 143.133,A -85,B 0,C 180,E1 -10961.761,E2 -10961.761} C_VEL
LIN {X 0,Y 404.204,Z 143.135,A -85,B 0,C 180,E1 -10964.881,E2 -10964.881} C_VEL
LIN {X 0,Y 404.255,Z 143.125,A -85,B 0,C 180,E1 -10967.958,E2 -10967.958} C_VEL
LIN {X 0,Y 404.403,Z 143.107,A -85,B 0,C 180,E1 -10972.128,E2 -10972.128} C_VEL
LIN {X 0,Y 404.418,Z 143.105,A -85,B 0,C 180,E1 -10974.014,E2 -10974.014} C_VEL
LIN {X 0,Y 404.481,Z 143.097,A -85,B 0,C 180,E1 -10978.008,E2 -10978.008} C_VEL
LIN {X 0,Y 404.61,Z 143.081,A -85,B 0,C 180,E1 -10979.999,E2 -10979.999} C_VEL
LIN {X 0,Y 404.42,Z 143.109,A -85,B 0,C 180,E1 -10982.988,E2 -10982.988} C_VEL
LIN {X 0,Y 404.397,Z 143.111,A -85,B 0,C 180,E1 -10986.987,E2 -10986.987} C_VEL
LIN {X 0,Y 404.256,Z 143.126,A -85,B 0,C 180,E1 -10990.011,E2 -10990.011} C_VEL
LIN {X 0,Y 404.263,Z 143.125,A -85,B 0,C 180,E1 -10993.211,E2 -10993.211} C_VEL
LIN {X 0,Y 404.212,Z 143.132,A -85,B 0,C 180,E1 -10997.007,E2 -10997.007} C_VEL
LIN {X 0,Y 404.183,Z 143.141,A -85,B 0,C 180,E1 -11000.35,E2 -11000.35} C_VEL
LIN {X 0,Y 404.166,Z 143.137,A -85,B 0,C 180,E1 -11003.574,E2 -11003.574} C_VEL
LIN {X 0,Y 404.179,Z 143.136,A -85,B 0,C 180,E1 -11005.766,E2 -11005.766} C_VEL
LIN {X 0,Y 404.191,Z 143.137,A -85,B 0,C 180,E1 -11007.999,E2 -11007.999} C_VEL
LIN {X 0,Y 404.135,Z 143.141,A -85,B 0,C 180,E1 -11011.558,E2 -11011.558} C_VEL
LIN {X 0,Y 404.181,Z 143.135,A -85,B 0,C 180,E1 -11015.016,E2 -11015.016} C_VEL
LIN {X 0,Y 404.159,Z 143.138,A -85,B 0,C 180,E1 -11018.756,E2 -11018.756} C_VEL
LIN {X 0,Y 404.187,Z 143.137,A -85,B 0,C 180,E1 -11021.611,E2 -11021.611} C_VEL
LIN {X 0,Y 404.196,Z 143.134,A -85,B 0,C 180,E1 -11024.53,E2 -11024.53} C_VEL
LIN {X 0,Y 404.206,Z 143.133,A -85,B 0,C 180,E1 -11027.305,E2 -11027.305} C_VEL
LIN {X 0,Y 404.164,Z 143.142,A -85,B 0,C 180,E1 -11029.956,E2 -11029.956} C_VEL
LIN {X 0,Y 404.136,Z 143.141,A -85,B 0,C 180,E1 -11033.124,E2 -11033.124} C_VEL
LIN {X 0,Y 404.14,Z 143.141,A -85,B 0,C 180,E1 -11036.188,E2 -11036.188} C_VEL
LIN {X 0,Y 404.14,Z 143.146,A -85,B 0,C 180,E1 -11039.715,E2 -11039.715} C_VEL
LIN {X 0,Y 404.19,Z 143.136,A -85,B 0,C 180,E1 -11043.123,E2 -11043.123} C_VEL
LIN {X 0,Y 404.173,Z 143.141,A -85,B 0,C 180,E1 -11045.335,E2 -11045.335} C_VEL
LIN {X 0,Y 404.134,Z 143.14,A -85,B 0,C 180,E1 -11048.581,E2 -11048.581} C_VEL
LIN {X 0,Y 404.206,Z 143.134,A -85,B 0,C 180,E1 -11051.762,E2 -11051.762} C_VEL
LIN {X 0,Y 404.202,Z 143.134,A -85,B 0,C 180,E1 -11054.882,E2 -11054.882} C_VEL
LIN {X 0,Y 404.253,Z 143.126,A -85,B 0,C 180,E1 -11057.959,E2 -11057.959} C_VEL
LIN {X 0,Y 404.429,Z 143.104,A -85,B 0,C 180,E1 -11062.1,E2 -11062.1} C_VEL
LIN {X 0,Y 404.421,Z 143.105,A -85,B 0,C 180,E1 -11064.016,E2 -11064.016} C_VEL
LIN {X 0,Y 404.479,Z 143.097,A -85,B 0,C 180,E1 -11068.009,E2 -11068.009} C_VEL
LIN {X 0,Y 404.608,Z 143.081,A -85,B 0,C 180,E1 -11070.001,E2 -11070.001} C_VEL
LIN {X 0,Y 404.42,Z 143.111,A -85,B 0,C 180,E1 -11072.989,E2 -11072.989} C_VEL
LIN {X 0,Y 404.409,Z 143.112,A -85,B 0,C 180,E1 -11076.988,E2 -11076.988} C_VEL
LIN {X 0,Y 404.256,Z 143.125,A -85,B 0,C 180,E1 -11080.012,E2 -11080.012} C_VEL
LIN {X 0,Y 404.25,Z 143.13,A -85,B 0,C 180,E1 -11083.204,E2 -11083.204} C_VEL
LIN {X 0,Y 404.307,Z 143.138,A -85,B 0,C 180,E1 -11086.149,E2 -11086.149} C_VEL
LIN {X 0,Y 405.974,Z 152.975,A -85,B 0,C 180,E1 -11088.548,E2 -11088.548} C_VEL
LIN {X 0,Y 408.345,Z 163.41,A -85,B 0,C 180,E1 -11088.858,E2 -11088.858} C_VEL
LIN {X 0,Y 408.633,Z 167.279,A -85,B 0,C 180,E1 -11088.945,E2 -11088.945} C_VEL
LIN {X 0,Y 408.29,Z 171.183,A -85,B 0,C 180,E1 -11089.004,E2 -11089.004} C_VEL
LIN {X 0,Y 406.468,Z 178.925,A -85,B 0,C 180,E1 -11089.071,E2 -11089.071} C_VEL
LIN {X 0,Y 404.265,Z 186.715,A -85,B 0,C 180,E1 -11089.123,E2 -11089.123} C_VEL
LIN {X 0,Y 403.238,Z 192.639,A -85,B 0,C 180,E1 -11089.191,E2 -11089.191} C_VEL
LIN {X 0,Y 403.138,Z 194.632,A -85,B 0,C 180,E1 -11089.225,E2 -11089.225} C_VEL
LIN {X 0,Y 402.031,Z 260.963,A -85,B 0,C 180,E1 -11090.482,E2 -11090.482} C_VEL
LIN {X 0,Y 401.626,Z 274.613,A -85,B 0,C 180,E1 -11090.956,E2 -11090.956} C_VEL
LIN {X 0,Y 401.136,Z 286.958,A -85,B 0,C 180,E1 -11091.588,E2 -11091.588} C_VEL
LIN {X 0,Y 400.523,Z 299.267,A -85,B 0,C 180,E1 -11092.448,E2 -11092.448} C_VEL
LIN {X 0,Y 399.709,Z 310.428,A -85,B 0,C 180,E1 -11093.442,E2 -11093.442} C_VEL
LIN {X 0,Y 398.978,Z 320.729,A -85,B 0,C 180,E1 -11094.593,E2 -11094.593} C_VEL
LIN {X 0,Y 398.23,Z 330.608,A -85,B 0,C 180,E1 -11095.973,E2 -11095.973} C_VEL
LIN {X 0,Y 397.59,Z 338.684,A -85,B 0,C 180,E1 -11097.361,E2 -11097.361} C_VEL
LIN {X 0,Y 397.053,Z 345.672,A -85,B 0,C 180,E1 -11098.839,E2 -11098.839} C_VEL
LIN {X 0,Y 396.594,Z 351.353,A -85,B 0,C 180,E1 -11100.334,E2 -11100.334} C_VEL
LIN {X 0,Y 396.215,Z 356.641,A -85,B 0,C 180,E1 -11102.151,E2 -11102.151} C_VEL
LIN {X 0,Y 396.008,Z 359.573,A -85,B 0,C 180,E1 -11103.478,E2 -11103.478} C_VEL
LIN {X 0,Y 395.756,Z 362.259,A -85,B 0,C 180,E1 -11105.227,E2 -11105.227} C_VEL
LIN {X 0,Y 395.656,Z 363.818,A -85,B 0,C 180,E1 -11107.153,E2 -11107.153} C_VEL
LIN {X 0,Y 395.671,Z 364.038,A -85,B 0,C 180,E1 -11108.599,E2 -11108.599} C_VEL
LIN {X 0,Y 395.752,Z 363.335,A -85,B 0,C 180,E1 -11110.217,E2 -11110.217} C_VEL
LIN {X 0,Y 395.952,Z 361.658,A -85,B 0,C 180,E1 -11111.8,E2 -11111.8} C_VEL
LIN {X 0,Y 396.242,Z 358.18,A -85,B 0,C 180,E1 -11113.768,E2 -11113.768} C_VEL
LIN {X 0,Y 396.517,Z 354.688,A -85,B 0,C 180,E1 -11115.152,E2 -11115.152} C_VEL
LIN {X 0,Y 397.04,Z 349.155,A -85,B 0,C 180,E1 -11116.852,E2 -11116.852} C_VEL
LIN {X 0,Y 397.709,Z 341.797,A -85,B 0,C 180,E1 -11118.583,E2 -11118.583} C_VEL
LIN {X 0,Y 398.421,Z 334.209,A -85,B 0,C 180,E1 -11120.009,E2 -11120.009} C_VEL
LIN {X 0,Y 399.161,Z 325.708,A -85,B 0,C 180,E1 -11121.315,E2 -11121.315} C_VEL
LIN {X 0,Y 399.994,Z 316.349,A -85,B 0,C 180,E1 -11122.486,E2 -11122.486} C_VEL
LIN {X 0,Y 400.896,Z 305.193,A -85,B 0,C 180,E1 -11123.604,E2 -11123.604} C_VEL
LIN {X 0,Y 401.707,Z 293.825,A -85,B 0,C 180,E1 -11124.506,E2 -11124.506} C_VEL
LIN {X 0,Y 402.357,Z 281.573,A -85,B 0,C 180,E1 -11125.25,E2 -11125.25} C_VEL
LIN {X 0,Y 402.817,Z 269.079,A -85,B 0,C 180,E1 -11125.794,E2 -11125.794} C_VEL
LIN {X 0,Y 403.22,Z 255.493,A -85,B 0,C 180,E1 -11126.164,E2 -11126.164} C_VEL
LIN {X 0,Y 404.606,Z 174.907,A -85,B 0,C 180,E1 -11127.689,E2 -11127.689} C_VEL
LIN {X 0,Y 401.288,Z 159.993,A -85,B 0,C 180,E1 -11128.184,E2 -11128.184} C_VEL
LIN {X 0,Y 399.253,Z 154.004,A -85,B 0,C 180,E1 -11128.458,E2 -11128.458} C_VEL
LIN {X 0,Y 397.134,Z 144.018,A -85,B 0,C 180,E1 -11131.024,E2 -11131.024} C_VEL
LIN {X 0,Y 397.136,Z 144.021,A -85,B 0,C 180,E1 -11133.742,E2 -11133.742} C_VEL
LIN {X 0,Y 397.107,Z 144.025,A -85,B 0,C 180,E1 -11137.086,E2 -11137.086} C_VEL
LIN {X 0,Y 397.15,Z 144.015,A -85,B 0,C 180,E1 -11140.354,E2 -11140.354} C_VEL
LIN {X 0,Y 397.17,Z 144.012,A -85,B 0,C 180,E1 -11143.554,E2 -11143.554} C_VEL
LIN {X 0,Y 397.233,Z 144.006,A -85,B 0,C 180,E1 -11146.703,E2 -11146.703} C_VEL
LIN {X 0,Y 397.22,Z 144.003,A -85,B 0,C 180,E1 -11149.81,E2 -11149.81} C_VEL
LIN {X 0,Y 397.298,Z 143.997,A -85,B 0,C 180,E1 -11152.888,E2 -11152.888} C_VEL
LIN {X 0,Y 397.238,Z 144.002,A -85,B 0,C 180,E1 -11154.926,E2 -11154.926} C_VEL
LIN {X 0,Y 397.445,Z 143.98,A -85,B 0,C 180,E1 -11157.974,E2 -11157.974} C_VEL
LIN {X 0,Y 397.442,Z 143.977,A -85,B 0,C 180,E1 -11162.027,E2 -11162.027} C_VEL
LIN {X 0,Y 397.332,Z 143.987,A -85,B 0,C 180,E1 -11166.093,E2 -11166.093} C_VEL
LIN {X 0,Y 397.231,Z 144.002,A -85,B 0,C 180,E1 -11169.163,E2 -11169.163} C_VEL
LIN {X 0,Y 397.211,Z 144.005,A -85,B 0,C 180,E1 -11172.259,E2 -11172.259} C_VEL
LIN {X 0,Y 397.113,Z 144.012,A -85,B 0,C 180,E1 -11175.395,E2 -11175.395} C_VEL
LIN {X 0,Y 397.077,Z 144.018,A -85,B 0,C 180,E1 -11178.578,E2 -11178.578} C_VEL
LIN {X 0,Y 397.09,Z 144.021,A -85,B 0,C 180,E1 -11181.819,E2 -11181.819} C_VEL
LIN {X 0,Y 397.105,Z 144.019,A -85,B 0,C 180,E1 -11185.136,E2 -11185.136} C_VEL
LIN {X 0,Y 397.064,Z 144.019,A -85,B 0,C 180,E1 -11188.549,E2 -11188.549} C_VEL
LIN {X 0,Y 397.081,Z 144.018,A -85,B 0,C 180,E1 -11191.835,E2 -11191.835} C_VEL
LIN {X 0,Y 397.125,Z 144.017,A -85,B 0,C 180,E1 -11194.494,E2 -11194.494} C_VEL
LIN {X 0,Y 397.097,Z 144.018,A -85,B 0,C 180,E1 -11198.276,E2 -11198.276} C_VEL
LIN {X 0,Y 397.056,Z 144.024,A -85,B 0,C 180,E1 -11201.976,E2 -11201.976} C_VEL
LIN {X 0,Y 397.091,Z 144.025,A -85,B 0,C 180,E1 -11205.069,E2 -11205.069} C_VEL
LIN {X 0,Y 397.059,Z 144.029,A -85,B 0,C 180,E1 -11208.023,E2 -11208.023} C_VEL
LIN {X 0,Y 397.097,Z 144.022,A -85,B 0,C 180,E1 -11211.724,E2 -11211.724} C_VEL
LIN {X 0,Y 397.13,Z 144.017,A -85,B 0,C 180,E1 -11215.506,E2 -11215.506} C_VEL
LIN {X 0,Y 397.083,Z 144.025,A -85,B 0,C 180,E1 -11219.117,E2 -11219.117} C_VEL
LIN {X 0,Y 397.148,Z 144.154,A -85,B 0,C 180,E1 -11220.806,E2 -11220.806} C_VEL
LIN {X 0,Y 399.933,Z 156.722,A -85,B 0,C 180,E1 -11223.667,E2 -11223.667} C_VEL
LIN {X 0,Y 400.756,Z 162.091,A -85,B 0,C 180,E1 -11224.832,E2 -11224.832} C_VEL
LIN {X 0,Y 399.513,Z 178.265,A -85,B 0,C 180,E1 -11228.048,E2 -11228.048} C_VEL
LIN {X 0,Y 399.031,Z 186.1,A -85,B 0,C 180,E1 -11229.592,E2 -11229.592} C_VEL
LIN {X 0,Y 402.923,Z 209.755,A -85,B 0,C 180,E1 -11230.292,E2 -11230.292} C_VEL
LIN {X 0,Y 403.958,Z 219.088,A -85,B 0,C 180,E1 -11230.536,E2 -11230.536} C_VEL
LIN {X 0,Y 402.712,Z 296.06,A -85,B 0,C 180,E1 -11232.02,E2 -11232.02} C_VEL
LIN {X 0,Y 402.018,Z 309.584,A -85,B 0,C 180,E1 -11232.481,E2 -11232.481} C_VEL
LIN {X 0,Y 401.216,Z 322.417,A -85,B 0,C 180,E1 -11233.134,E2 -11233.134} C_VEL
LIN {X 0,Y 400.378,Z 334.182,A -85,B 0,C 180,E1 -11233.95,E2 -11233.95} C_VEL
LIN {X 0,Y 399.431,Z 345.568,A -85,B 0,C 180,E1 -11234.957,E2 -11234.957} C_VEL
LIN {X 0,Y 398.553,Z 356.374,A -85,B 0,C 180,E1 -11236.164,E2 -11236.164} C_VEL
LIN {X 0,Y 397.744,Z 365.964,A -85,B 0,C 180,E1 -11237.499,E2 -11237.499} C_VEL
LIN {X 0,Y 396.897,Z 374.876,A -85,B 0,C 180,E1 -11239.026,E2 -11239.026} C_VEL
LIN {X 0,Y 396.411,Z 382.018,A -85,B 0,C 180,E1 -11240.561,E2 -11240.561} C_VEL
LIN {X 0,Y 396.04,Z 388.568,A -85,B 0,C 180,E1 -11242.351,E2 -11242.351} C_VEL
LIN {X 0,Y 395.824,Z 392.893,A -85,B 0,C 180,E1 -11243.884,E2 -11243.884} C_VEL
LIN {X 0,Y 395.827,Z 395.199,A -85,B 0,C 180,E1 -11244.906,E2 -11244.906} C_VEL
LIN {X 0,Y 395.78,Z 397.018,A -85,B 0,C 180,E1 -11245.926,E2 -11245.926} C_VEL
LIN {X 0,Y 395.859,Z 399.396,A -85,B 0,C 180,E1 -11247.965,E2 -11247.965} C_VEL
LIN {X 0,Y 395.835,Z 399.984,A -85,B 0,C 180,E1 -11248.982,E2 -11248.982} C_VEL
LIN {X 0,Y 395.826,Z 400.129,A -85,B 0,C 180,E1 -11249.999,E2 -11249.999} C_VEL
LIN {X 0,Y 395.835,Z 399.87,A -85,B 0,C 180,E1 -11251.017,E2 -11251.017} C_VEL
LIN {X 0,Y 395.859,Z 399.218,A -85,B 0,C 180,E1 -11252.034,E2 -11252.034} C_VEL
LIN {X 0,Y 395.777,Z 398.158,A -85,B 0,C 180,E1 -11253.053,E2 -11253.053} C_VEL
LIN {X 0,Y 395.785,Z 396.638,A -85,B 0,C 180,E1 -11254.072,E2 -11254.072} C_VEL
LIN {X 0,Y 395.809,Z 393.125,A -85,B 0,C 180,E1 -11255.776,E2 -11255.776} C_VEL
LIN {X 0,Y 396.036,Z 387.749,A -85,B 0,C 180,E1 -11257.648,E2 -11257.648} C_VEL
LIN {X 0,Y 396.389,Z 380.835,A -85,B 0,C 180,E1 -11259.439,E2 -11259.439} C_VEL
LIN {X 0,Y 396.84,Z 373.315,A -85,B 0,C 180,E1 -11260.974,E2 -11260.974} C_VEL
LIN {X 0,Y 397.508,Z 365.654,A -85,B 0,C 180,E1 -11262.248,E2 -11262.248} C_VEL
LIN {X 0,Y 398.167,Z 357.042,A -85,B 0,C 180,E1 -11263.436,E2 -11263.436} C_VEL
LIN {X 0,Y 398.866,Z 347.291,A -85,B 0,C 180,E1 -11264.541,E2 -11264.541} C_VEL
LIN {X 0,Y 399.642,Z 336.106,A -85,B 0,C 180,E1 -11265.556,E2 -11265.556} C_VEL
LIN {X 0,Y 400.497,Z 323.596,A -85,B 0,C 180,E1 -11266.437,E2 -11266.437} C_VEL
LIN {X 0,Y 401.203,Z 310.896,A -85,B 0,C 180,E1 -11267.095,E2 -11267.095} C_VEL
LIN {X 0,Y 401.803,Z 297.519,A -85,B 0,C 180,E1 -11267.56,E2 -11267.56} C_VEL
LIN {X 0,Y 402.406,Z 261.761,A -85,B 0,C 180,E1 -11268.256,E2 -11268.256} C_VEL
LIN {X 0,Y 402.841,Z 216.38,A -85,B 0,C 180,E1 -11269.113,E2 -11269.113} C_VEL
LIN {X 0,Y 398.699,Z 187.293,A -85,B 0,C 180,E1 -11269.902,E2 -11269.902} C_VEL
LIN {X 0,Y 400.192,Z 166.398,A -85,B 0,C 180,E1 -11274.047,E2 -11274.047} C_VEL
LIN {X 0,Y 400.469,Z 160.748,A -85,B 0,C 180,E1 -11275.186,E2 -11275.186} C_VEL
LIN {X 0,Y 398.024,Z 147.845,A -85,B 0,C 180,E1 -11278.01,E2 -11278.01} C_VEL
LIN {X 0,Y 397.178,Z 144.013,A -85,B 0,C 180,E1 -11278.9,E2 -11278.9} C_VEL
LIN {X 0,Y 397.08,Z 144.026,A -85,B 0,C 180,E1 -11282.071,E2 -11282.071} C_VEL
LIN {X 0,Y 397.12,Z 144.016,A -85,B 0,C 180,E1 -11285.503,E2 -11285.503} C_VEL
LIN {X 0,Y 397.132,Z 144.013,A -85,B 0,C 180,E1 -11288.861,E2 -11288.861} C_VEL
LIN {X 0,Y 397.069,Z 144.023,A -85,B 0,C 180,E1 -11292.266,E2 -11292.266} C_VEL
LIN {X 0,Y 397.087,Z 144.019,A -85,B 0,C 180,E1 -11295.068,E2 -11295.068} C_VEL
LIN {X 0,Y 397.066,Z 144.024,A -85,B 0,C 180,E1 -11298.02,E2 -11298.02} C_VEL
LIN {X 0,Y 397.126,Z 144.015,A -85,B 0,C 180,E1 -11301.139,E2 -11301.139} C_VEL
LIN {X 0,Y 397.118,Z 144.014,A -85,B 0,C 180,E1 -11304.496,E2 -11304.496} C_VEL
LIN {X 0,Y 397.077,Z 144.022,A -85,B 0,C 180,E1 -11307.928,E2 -11307.928} C_VEL
LIN {X 0,Y 397.122,Z 144.021,A -85,B 0,C 180,E1 -11311.456,E2 -11311.456} C_VEL
LIN {X 0,Y 397.152,Z 144.01,A -85,B 0,C 180,E1 -11314.487,E2 -11314.487} C_VEL
LIN {X 0,Y 397.108,Z 144.02,A -85,B 0,C 180,E1 -11317.085,E2 -11317.085} C_VEL
LIN {X 0,Y 397.145,Z 144.011,A -85,B 0,C 180,E1 -11320.352,E2 -11320.352} C_VEL
LIN {X 0,Y 397.165,Z 144.011,A -85,B 0,C 180,E1 -11323.553,E2 -11323.553} C_VEL
LIN {X 0,Y 397.227,Z 144.003,A -85,B 0,C 180,E1 -11326.702,E2 -11326.702} C_VEL
LIN {X 0,Y 397.216,Z 144.003,A -85,B 0,C 180,E1 -11329.808,E2 -11329.808} C_VEL
LIN {X 0,Y 397.348,Z 143.992,A -85,B 0,C 180,E1 -11332.887,E2 -11332.887} C_VEL
LIN {X 0,Y 397.252,Z 144.005,A -85,B 0,C 180,E1 -11334.925,E2 -11334.925} C_VEL
LIN {X 0,Y 397.45,Z 143.973,A -85,B 0,C 180,E1 -11337.973,E2 -11337.973} C_VEL
LIN {X 0,Y 397.579,Z 143.957,A -85,B 0,C 180,E1 -11339.999,E2 -11339.999} C_VEL
LIN {X 0,Y 397.378,Z 143.986,A -85,B 0,C 180,E1 -11343.041,E2 -11343.041} C_VEL
LIN {X 0,Y 397.342,Z 143.986,A -85,B 0,C 180,E1 -11346.577,E2 -11346.577} C_VEL
LIN {X 0,Y 397.25,Z 144,A -85,B 0,C 180,E1 -11349.161,E2 -11349.161} C_VEL
LIN {X 0,Y 397.216,Z 144.005,A -85,B 0,C 180,E1 -11352.258,E2 -11352.258} C_VEL
LIN {X 0,Y 397.176,Z 144.007,A -85,B 0,C 180,E1 -11355.392,E2 -11355.392} C_VEL
LIN {X 0,Y 397.159,Z 144.015,A -85,B 0,C 180,E1 -11358.573,E2 -11358.573} C_VEL
LIN {X 0,Y 397.093,Z 144.019,A -85,B 0,C 180,E1 -11361.818,E2 -11361.818} C_VEL
LIN {X 0,Y 397.152,Z 144.01,A -85,B 0,C 180,E1 -11365.131,E2 -11365.131} C_VEL
LIN {X 0,Y 397.158,Z 144.011,A -85,B 0,C 180,E1 -11367.776,E2 -11367.776} C_VEL
LIN {X 0,Y 397.074,Z 144.021,A -85,B 0,C 180,E1 -11370.882,E2 -11370.882} C_VEL
LIN {X 0,Y 397.121,Z 144.017,A -85,B 0,C 180,E1 -11374.493,E2 -11374.493} C_VEL
LIN {X 0,Y 397.105,Z 144.02,A -85,B 0,C 180,E1 -11378.274,E2 -11378.274} C_VEL
LIN {X 0,Y 397.152,Z 144.017,A -85,B 0,C 180,E1 -11381.993,E2 -11381.993} C_VEL
LIN {X 0,Y 397.146,Z 144.011,A -85,B 0,C 180,E1 -11385.059,E2 -11385.059} C_VEL
LIN {X 0,Y 397.151,Z 144.015,A -85,B 0,C 180,E1 -11388.007,E2 -11388.007} C_VEL
LIN {X 0,Y 397.105,Z 144.022,A -85,B 0,C 180,E1 -11391.726,E2 -11391.726} C_VEL
LIN {X 0,Y 397.121,Z 144.019,A -85,B 0,C 180,E1 -11395.507,E2 -11395.507} C_VEL
LIN {X 0,Y 397.073,Z 144.022,A -85,B 0,C 180,E1 -11399.118,E2 -11399.118} C_VEL
LIN {X 0,Y 397.189,Z 144.006,A -85,B 0,C 180,E1 -11402.61,E2 -11402.61} C_VEL
LIN {X 0,Y 397.128,Z 144.015,A -85,B 0,C 180,E1 -11405.982,E2 -11405.982} C_VEL
LIN {X 0,Y 397.134,Z 144.016,A -85,B 0,C 180,E1 -11409.705,E2 -11409.705} C_VEL
LIN {X 0,Y 397.177,Z 144.009,A -85,B 0,C 180,E1 -11412.845,E2 -11412.845} C_VEL
LIN {X 0,Y 397.222,Z 144.003,A -85,B 0,C 180,E1 -11416.679,E2 -11416.679} C_VEL
LIN {X 0,Y 397.214,Z 144.004,A -85,B 0,C 180,E1 -11419.809,E2 -11419.809} C_VEL
LIN {X 0,Y 397.36,Z 143.988,A -85,B 0,C 180,E1 -11422.889,E2 -11422.889} C_VEL
LIN {X 0,Y 397.252,Z 144.002,A -85,B 0,C 180,E1 -11424.926,E2 -11424.926} C_VEL
LIN {X 0,Y 397.448,Z 143.973,A -85,B 0,C 180,E1 -11427.974,E2 -11427.974} C_VEL
LIN {X 0,Y 397.578,Z 143.957,A -85,B 0,C 180,E1 -11430.001,E2 -11430.001} C_VEL
LIN {X 0,Y 397.378,Z 143.988,A -85,B 0,C 180,E1 -11433.042,E2 -11433.042} C_VEL
LIN {X 0,Y 397.361,Z 143.988,A -85,B 0,C 180,E1 -11437.112,E2 -11437.112} C_VEL
LIN {X 0,Y 397.216,Z 144.003,A -85,B 0,C 180,E1 -11440.192,E2 -11440.192} C_VEL
LIN {X 0,Y 397.205,Z 144.007,A -85,B 0,C 180,E1 -11443.311,E2 -11443.311} C_VEL
LIN {X 0,Y 397.255,Z 144.107,A -85,B 0,C 180,E1 -11445.949,E2 -11445.949} C_VEL
LIN {X 0,Y 398.943,Z 153.415,A -85,B 0,C 180,E1 -11448.225,E2 -11448.225} C_VEL
LIN {X 0,Y 401.734,Z 165.038,A -85,B 0,C 180,E1 -11448.586,E2 -11448.586} C_VEL
LIN {X 0,Y 403.424,Z 173.781,A -85,B 0,C 180,E1 -11448.835,E2 -11448.835} C_VEL
LIN {X 0,Y 403.138,Z 194.632,A -85,B 0,C 180,E1 -11449.225,E2 -11449.225} C_VEL
LIN {X 0,Y 402.401,Z 200.473,A -85,B 0,C 180,E1 -11449.305,E2 -11449.305} C_VEL
LIN {X 0,Y 396.467,Z 219.415,A -85,B 0,C 180,E1 -11449.411,E2 -11449.411} C_VEL
LIN {X 0,Y 395.807,Z 225.253,A -85,B 0,C 180,E1 -11449.496,E2 -11449.496} C_VEL
LIN {X 0,Y 395.221,Z 261.856,A -85,B 0,C 180,E1 -11450.222,E2 -11450.222} C_VEL
LIN {X 0,Y 394.779,Z 275.741,A -85,B 0,C 180,E1 -11450.722,E2 -11450.722} C_VEL
LIN {X 0,Y 394.252,Z 287.843,A -85,B 0,C 180,E1 -11451.367,E2 -11451.367} C_VEL
LIN {X 0,Y 393.701,Z 298.961,A -85,B 0,C 180,E1 -11452.155,E2 -11452.155} C_VEL
LIN {X 0,Y 392.82,Z 310.386,A -85,B 0,C 180,E1 -11453.18,E2 -11453.18} C_VEL
LIN {X 0,Y 392.058,Z 320.764,A -85,B 0,C 180,E1 -11454.35,E2 -11454.35} C_VEL
LIN {X 0,Y 391.371,Z 329.288,A -85,B 0,C 180,E1 -11455.53,E2 -11455.53} C_VEL
LIN {X 0,Y 390.654,Z 338.033,A -85,B 0,C 180,E1 -11457.018,E2 -11457.018} C_VEL
LIN {X 0,Y 390.058,Z 345.296,A -85,B 0,C 180,E1 -11458.545,E2 -11458.545} C_VEL
LIN {X 0,Y 389.504,Z 352.053,A -85,B 0,C 180,E1 -11460.346,E2 -11460.346} C_VEL
LIN {X 0,Y 389.176,Z 356.596,A -85,B 0,C 180,E1 -11461.925,E2 -11461.925} C_VEL
LIN {X 0,Y 388.863,Z 360.483,A -85,B 0,C 180,E1 -11463.762,E2 -11463.762} C_VEL
LIN {X 0,Y 388.648,Z 362.951,A -85,B 0,C 180,E1 -11465.538,E2 -11465.538} C_VEL
LIN {X 0,Y 388.573,Z 364.193,A -85,B 0,C 180,E1 -11467.269,E2 -11467.269} C_VEL
LIN {X 0,Y 388.599,Z 364.224,A -85,B 0,C 180,E1 -11469.272,E2 -11469.272} C_VEL
LIN {X 0,Y 388.709,Z 363.421,A -85,B 0,C 180,E1 -11470.61,E2 -11470.61} C_VEL
LIN {X 0,Y 388.914,Z 361.582,A -85,B 0,C 180,E1 -11472.193,E2 -11472.193} C_VEL
LIN {X 0,Y 389.156,Z 358.815,A -85,B 0,C 180,E1 -11473.749,E2 -11473.749} C_VEL
LIN {X 0,Y 389.482,Z 355.113,A -85,B 0,C 180,E1 -11475.274,E2 -11475.274} C_VEL
LIN {X 0,Y 389.951,Z 350.401,A -85,B 0,C 180,E1 -11476.776,E2 -11476.776} C_VEL
LIN {X 0,Y 390.505,Z 344.623,A -85,B 0,C 180,E1 -11478.25,E2 -11478.25} C_VEL
LIN {X 0,Y 391.198,Z 337.606,A -85,B 0,C 180,E1 -11479.704,E2 -11479.704} C_VEL
LIN {X 0,Y 392.025,Z 329.066,A -85,B 0,C 180,E1 -11481.138,E2 -11481.138} C_VEL
LIN {X 0,Y 393.033,Z 318.478,A -85,B 0,C 180,E1 -11482.558,E2 -11482.558} C_VEL
LIN {X 0,Y 393.916,Z 307.833,A -85,B 0,C 180,E1 -11483.702,E2 -11483.702} C_VEL
LIN {X 0,Y 394.849,Z 296.655,A -85,B 0,C 180,E1 -11484.642,E2 -11484.642} C_VEL
LIN {X 0,Y 395.552,Z 284.794,A -85,B 0,C 180,E1 -11485.421,E2 -11485.421} C_VEL
LIN {X 0,Y 396.051,Z 272.314,A -85,B 0,C 180,E1 -11486.028,E2 -11486.028} C_VEL
LIN {X 0,Y 396.445,Z 259.611,A -85,B 0,C 180,E1 -11486.43,E2 -11486.43} C_VEL
LIN {X 0,Y 398.02,Z 175.745,A -85,B 0,C 180,E1 -11488.055,E2 -11488.055} C_VEL
LIN {X 0,Y 394.784,Z 161.533,A -85,B 0,C 180,E1 -11488.546,E2 -11488.546} C_VEL
LIN {X 0,Y 392.134,Z 154.461,A -85,B 0,C 180,E1 -11488.872,E2 -11488.872} C_VEL
LIN {X 0,Y 390.095,Z 144.893,A -85,B 0,C 180,E1 -11491.41,E2 -11491.41} C_VEL
LIN {X 0,Y 390.112,Z 144.896,A -85,B 0,C 180,E1 -11494.383,E2 -11494.383} C_VEL
LIN {X 0,Y 390.04,Z 144.903,A -85,B 0,C 180,E1 -11497.767,E2 -11497.767} C_VEL
LIN {X 0,Y 390.106,Z 144.894,A -85,B 0,C 180,E1 -11501.079,E2 -11501.079} C_VEL
LIN {X 0,Y 390.142,Z 144.888,A -85,B 0,C 180,E1 -11504.324,E2 -11504.324} C_VEL
LIN {X 0,Y 390.175,Z 144.885,A -85,B 0,C 180,E1 -11507.518,E2 -11507.518} C_VEL
LIN {X 0,Y 390.197,Z 144.886,A -85,B 0,C 180,E1 -11510.672,E2 -11510.672} C_VEL
LIN {X 0,Y 390.287,Z 144.87,A -85,B 0,C 180,E1 -11513.798,E2 -11513.798} C_VEL
LIN {X 0,Y 390.412,Z 144.856,A -85,B 0,C 180,E1 -11517.937,E2 -11517.937} C_VEL
LIN {X 0,Y 390.408,Z 144.852,A -85,B 0,C 180,E1 -11522.064,E2 -11522.064} C_VEL
LIN {X 0,Y 390.286,Z 144.863,A -85,B 0,C 180,E1 -11526.203,E2 -11526.203} C_VEL
LIN {X 0,Y 390.189,Z 144.88,A -85,B 0,C 180,E1 -11529.33,E2 -11529.33} C_VEL
LIN {X 0,Y 390.158,Z 144.882,A -85,B 0,C 180,E1 -11532.484,E2 -11532.484} C_VEL
LIN {X 0,Y 390.057,Z 144.892,A -85,B 0,C 180,E1 -11535.681,E2 -11535.681} C_VEL
LIN {X 0,Y 390.035,Z 144.896,A -85,B 0,C 180,E1 -11538.926,E2 -11538.926} C_VEL
LIN {X 0,Y 390.034,Z 144.898,A -85,B 0,C 180,E1 -11542.235,E2 -11542.235} C_VEL
LIN {X 0,Y 390.055,Z 144.898,A -85,B 0,C 180,E1 -11545.722,E2 -11545.722} C_VEL
LIN {X 0,Y 390.026,Z 144.901,A -85,B 0,C 180,E1 -11549.113,E2 -11549.113} C_VEL
LIN {X 0,Y 390.045,Z 144.897,A -85,B 0,C 180,E1 -11552.722,E2 -11552.722} C_VEL
LIN {X 0,Y 390.059,Z 144.895,A -85,B 0,C 180,E1 -11555.825,E2 -11555.825} C_VEL
LIN {X 0,Y 390.042,Z 144.901,A -85,B 0,C 180,E1 -11559.212,E2 -11559.212} C_VEL
LIN {X 0,Y 390.035,Z 144.901,A -85,B 0,C 180,E1 -11562.372,E2 -11562.372} C_VEL
LIN {X 0,Y 390.048,Z 144.901,A -85,B 0,C 180,E1 -11565.354,E2 -11565.354} C_VEL
LIN {X 0,Y 390.022,Z 144.907,A -85,B 0,C 180,E1 -11568.185,E2 -11568.185} C_VEL
LIN {X 0,Y 390.064,Z 144.898,A -85,B 0,C 180,E1 -11570.904,E2 -11570.904} C_VEL
LIN {X 0,Y 390.09,Z 144.895,A -85,B 0,C 180,E1 -11574.793,E2 -11574.793} C_VEL
LIN {X 0,Y 390.029,Z 144.908,A -85,B 0,C 180,E1 -11578.495,E2 -11578.495} C_VEL
LIN {X 0,Y 390.116,Z 145.095,A -85,B 0,C 180,E1 -11580.45,E2 -11580.45} C_VEL
LIN {X 0,Y 392.961,Z 157.911,A -85,B 0,C 180,E1 -11583.44,E2 -11583.44} C_VEL
LIN {X 0,Y 393.853,Z 163.322,A -85,B 0,C 180,E1 -11584.642,E2 -11584.642} C_VEL
LIN {X 0,Y 392.698,Z 178.128,A -85,B 0,C 180,E1 -11587.647,E2 -11587.647} C_VEL
LIN {X 0,Y 392.178,Z 185.693,A -85,B 0,C 180,E1 -11589.168,E2 -11589.168} C_VEL
LIN {X 0,Y 396.191,Z 209.667,A -85,B 0,C 180,E1 -11589.91,E2 -11589.91} C_VEL
LIN {X 0,Y 397.332,Z 218.717,A -85,B 0,C 180,E1 -11590.16,E2 -11590.16} C_VEL
LIN {X 0,Y 396.047,Z 295.727,A -85,B 0,C 180,E1 -11591.673,E2 -11591.673} C_VEL
LIN {X 0,Y 395.323,Z 309.228,A -85,B 0,C 180,E1 -11592.141,E2 -11592.141} C_VEL
LIN {X 0,Y 394.518,Z 321.53,A -85,B 0,C 180,E1 -11592.772,E2 -11592.772} C_VEL
LIN {X 0,Y 393.56,Z 334.186,A -85,B 0,C 180,E1 -11593.664,E2 -11593.664} C_VEL
LIN {X 0,Y 392.554,Z 345.492,A -85,B 0,C 180,E1 -11594.687,E2 -11594.687} C_VEL
LIN {X 0,Y 391.678,Z 355.75,A -85,B 0,C 180,E1 -11595.853,E2 -11595.853} C_VEL
LIN {X 0,Y 390.949,Z 364.13,A -85,B 0,C 180,E1 -11597.014,E2 -11597.014} C_VEL
LIN {X 0,Y 390.021,Z 373.293,A -85,B 0,C 180,E1 -11598.567,E2 -11598.567} C_VEL
LIN {X 0,Y 389.447,Z 380.699,A -85,B 0,C 180,E1 -11600.128,E2 -11600.128} C_VEL
LIN {X 0,Y 389.063,Z 386.647,A -85,B 0,C 180,E1 -11601.69,E2 -11601.69} C_VEL
LIN {X 0,Y 388.825,Z 391.34,A -85,B 0,C 180,E1 -11603.252,E2 -11603.252} C_VEL
LIN {X 0,Y 388.721,Z 394.922,A -85,B 0,C 180,E1 -11604.813,E2 -11604.813} C_VEL
LIN {X 0,Y 388.703,Z 396.727,A -85,B 0,C 180,E1 -11605.852,E2 -11605.852} C_VEL
LIN {X 0,Y 388.757,Z 399.09,A -85,B 0,C 180,E1 -11607.927,E2 -11607.927} C_VEL
LIN {X 0,Y 388.764,Z 399.668,A -85,B 0,C 180,E1 -11608.964,E2 -11608.964} C_VEL
LIN {X 0,Y 388.753,Z 399.799,A -85,B 0,C 180,E1 -11609.999,E2 -11609.999} C_VEL
LIN {X 0,Y 388.764,Z 399.532,A -85,B 0,C 180,E1 -11611.035,E2 -11611.035} C_VEL
LIN {X 0,Y 388.772,Z 398.87,A -85,B 0,C 180,E1 -11612.071,E2 -11612.071} C_VEL
LIN {X 0,Y 388.68,Z 397.796,A -85,B 0,C 180,E1 -11613.109,E2 -11613.109} C_VEL
LIN {X 0,Y 388.709,Z 396.262,A -85,B 0,C 180,E1 -11614.147,E2 -11614.147} C_VEL
LIN {X 0,Y 388.711,Z 393.099,A -85,B 0,C 180,E1 -11615.727,E2 -11615.727} C_VEL
LIN {X 0,Y 388.898,Z 388.958,A -85,B 0,C 180,E1 -11617.267,E2 -11617.267} C_VEL
LIN {X 0,Y 389.191,Z 382.541,A -85,B 0,C 180,E1 -11619.091,E2 -11619.091} C_VEL
LIN {X 0,Y 389.621,Z 375.538,A -85,B 0,C 180,E1 -11620.654,E2 -11620.654} C_VEL
LIN {X 0,Y 390.388,Z 366.758,A -85,B 0,C 180,E1 -11622.211,E2 -11622.211} C_VEL
LIN {X 0,Y 391.095,Z 357.75,A -85,B 0,C 180,E1 -11623.509,E2 -11623.509} C_VEL
LIN {X 0,Y 391.855,Z 347.85,A -85,B 0,C 180,E1 -11624.674,E2 -11624.674} C_VEL
LIN {X 0,Y 392.659,Z 336.939,A -85,B 0,C 180,E1 -11625.706,E2 -11625.706} C_VEL
LIN {X 0,Y 393.52,Z 324.718,A -85,B 0,C 180,E1 -11626.603,E2 -11626.603} C_VEL
LIN {X 0,Y 394.28,Z 311.963,A -85,B 0,C 180,E1 -11627.304,E2 -11627.304} C_VEL
LIN {X 0,Y 394.881,Z 299.325,A -85,B 0,C 180,E1 -11627.778,E2 -11627.778} C_VEL
LIN {X 0,Y 395.29,Z 281.904,A -85,B 0,C 180,E1 -11628.161,E2 -11628.161} C_VEL
LIN {X 0,Y 396.083,Z 217.152,A -85,B 0,C 180,E1 -11629.398,E2 -11629.398} C_VEL
LIN {X 0,Y 391.764,Z 187.163,A -85,B 0,C 180,E1 -11630.202,E2 -11630.202} C_VEL
LIN {X 0,Y 393.298,Z 166.819,A -85,B 0,C 180,E1 -11634.308,E2 -11634.308} C_VEL
LIN {X 0,Y 393.475,Z 161.62,A -85,B 0,C 180,E1 -11635.383,E2 -11635.383} C_VEL
LIN {X 0,Y 390.971,Z 148.728,A -85,B 0,C 180,E1 -11638.259,E2 -11638.259} C_VEL
LIN {X 0,Y 390.121,Z 144.892,A -85,B 0,C 180,E1 -11639.178,E2 -11639.178} C_VEL
LIN {X 0,Y 390.044,Z 144.899,A -85,B 0,C 180,E1 -11642.721,E2 -11642.721} C_VEL
LIN {X 0,Y 390.057,Z 144.899,A -85,B 0,C 180,E1 -11645.825,E2 -11645.825} C_VEL
LIN {X 0,Y 390.071,Z 144.893,A -85,B 0,C 180,E1 -11649.218,E2 -11649.218} C_VEL
LIN {X 0,Y 390.043,Z 144.897,A -85,B 0,C 180,E1 -11652.373,E2 -11652.373} C_VEL
LIN {X 0,Y 390.044,Z 144.898,A -85,B 0,C 180,E1 -11655.354,E2 -11655.354} C_VEL
LIN {X 0,Y 390.031,Z 144.899,A -85,B 0,C 180,E1 -11658.186,E2 -11658.186} C_VEL
LIN {X 0,Y 390.087,Z 144.891,A -85,B 0,C 180,E1 -11660.907,E2 -11660.907} C_VEL
LIN {X 0,Y 390.084,Z 144.891,A -85,B 0,C 180,E1 -11664.792,E2 -11664.792} C_VEL
LIN {X 0,Y 390.022,Z 144.898,A -85,B 0,C 180,E1 -11668.495,E2 -11668.495} C_VEL
LIN {X 0,Y 390.116,Z 144.887,A -85,B 0,C 180,E1 -11672.069,E2 -11672.069} C_VEL
LIN {X 0,Y 390.08,Z 144.896,A -85,B 0,C 180,E1 -11675.519,E2 -11675.519} C_VEL
LIN {X 0,Y 390.054,Z 144.897,A -85,B 0,C 180,E1 -11678.877,E2 -11678.877} C_VEL
LIN {X 0,Y 390.11,Z 144.887,A -85,B 0,C 180,E1 -11682.165,E2 -11682.165} C_VEL
LIN {X 0,Y 390.142,Z 144.887,A -85,B 0,C 180,E1 -11685.392,E2 -11685.392} C_VEL
LIN {X 0,Y 390.147,Z 144.885,A -85,B 0,C 180,E1 -11688.571,E2 -11688.571} C_VEL
LIN {X 0,Y 390.305,Z 144.863,A -85,B 0,C 180,E1 -11692.031,E2 -11692.031} C_VEL
LIN {X 0,Y 390.224,Z 144.879,A -85,B 0,C 180,E1 -11694.833,E2 -11694.833} C_VEL
LIN {X 0,Y 390.419,Z 144.849,A -85,B 0,C 180,E1 -11697.936,E2 -11697.936} C_VEL
LIN {X 0,Y 390.548,Z 144.833,A -85,B 0,C 180,E1 -11699.999,E2 -11699.999} C_VEL
LIN {X 0,Y 390.312,Z 144.866,A -85,B 0,C 180,E1 -11703.096,E2 -11703.096} C_VEL
LIN {X 0,Y 390.299,Z 144.864,A -85,B 0,C 180,E1 -11706.571,E2 -11706.571} C_VEL
LIN {X 0,Y 390.202,Z 144.877,A -85,B 0,C 180,E1 -11709.328,E2 -11709.328} C_VEL
LIN {X 0,Y 390.191,Z 144.877,A -85,B 0,C 180,E1 -11713.438,E2 -11713.438} C_VEL
LIN {X 0,Y 390.145,Z 144.883,A -85,B 0,C 180,E1 -11717.307,E2 -11717.307} C_VEL
LIN {X 0,Y 390.089,Z 144.896,A -85,B 0,C 180,E1 -11720.472,E2 -11720.472} C_VEL
LIN {X 0,Y 390.085,Z 144.89,A -85,B 0,C 180,E1 -11723.35,E2 -11723.35} C_VEL
LIN {X 0,Y 390.109,Z 144.889,A -85,B 0,C 180,E1 -11726.768,E2 -11726.768} C_VEL
LIN {X 0,Y 390.034,Z 144.903,A -85,B 0,C 180,E1 -11730.299,E2 -11730.299} C_VEL
LIN {X 0,Y 390.063,Z 144.899,A -85,B 0,C 180,E1 -11734.024,E2 -11734.024} C_VEL
LIN {X 0,Y 390.043,Z 144.897,A -85,B 0,C 180,E1 -11737.551,E2 -11737.551} C_VEL
LIN {X 0,Y 390.078,Z 144.892,A -85,B 0,C 180,E1 -11740.826,E2 -11740.826} C_VEL
LIN {X 0,Y 390.124,Z 144.892,A -85,B 0,C 180,E1 -11743.897,E2 -11743.897} C_VEL
LIN {X 0,Y 390.113,Z 144.887,A -85,B 0,C 180,E1 -11746.798,E2 -11746.798} C_VEL
LIN {X 0,Y 390.073,Z 144.896,A -85,B 0,C 180,E1 -11749.563,E2 -11749.563} C_VEL
LIN {X 0,Y 390.042,Z 144.897,A -85,B 0,C 180,E1 -11752.448,E2 -11752.448} C_VEL
LIN {X 0,Y 390.079,Z 144.894,A -85,B 0,C 180,E1 -11756.047,E2 -11756.047} C_VEL
LIN {X 0,Y 390.041,Z 144.9,A -85,B 0,C 180,E1 -11759.869,E2 -11759.869} C_VEL
LIN {X 0,Y 390.108,Z 144.891,A -85,B 0,C 180,E1 -11763.232,E2 -11763.232} C_VEL
LIN {X 0,Y 390.101,Z 144.889,A -85,B 0,C 180,E1 -11766.751,E2 -11766.751} C_VEL
LIN {X 0,Y 390.099,Z 144.89,A -85,B 0,C 180,E1 -11769.983,E2 -11769.983} C_VEL
LIN {X 0,Y 390.133,Z 144.89,A -85,B 0,C 180,E1 -11773.249,E2 -11773.249} C_VEL
LIN {X 0,Y 390.19,Z 144.878,A -85,B 0,C 180,E1 -11776.562,E2 -11776.562} C_VEL
LIN {X 0,Y 390.201,Z 144.878,A -85,B 0,C 180,E1 -11780.672,E2 -11780.672} C_VEL
LIN {X 0,Y 390.315,Z 144.865,A -85,B 0,C 180,E1 -11782.76,E2 -11782.76} C_VEL
LIN {X 0,Y 390.224,Z 144.877,A -85,B 0,C 180,E1 -11784.834,E2 -11784.834} C_VEL
LIN {X 0,Y 390.417,Z 144.849,A -85,B 0,C 180,E1 -11787.937,E2 -11787.937} C_VEL
LIN {X 0,Y 390.547,Z 144.833,A -85,B 0,C 180,E1 -11790.001,E2 -11790.001} C_VEL
LIN {X 0,Y 390.312,Z 144.867,A -85,B 0,C 180,E1 -11793.097,E2 -11793.097} C_VEL
LIN {X 0,Y 390.328,Z 144.861,A -85,B 0,C 180,E1 -11796.203,E2 -11796.203} C_VEL
LIN {X 0,Y 390.311,Z 144.864,A -85,B 0,C 180,E1 -11798.283,E2 -11798.283} C_VEL
LIN {X 0,Y 390.164,Z 144.885,A -85,B 0,C 180,E1 -11802.484,E2 -11802.484} C_VEL
LIN {X 0,Y 390.187,Z 144.97,A -85,B 0,C 180,E1 -11805.709,E2 -11805.709} C_VEL
LIN {X 0,Y 391.804,Z 153.453,A -85,B 0,C 180,E1 -11807.874,E2 -11807.874} C_VEL
LIN {X 0,Y 394.365,Z 163.228,A -85,B 0,C 180,E1 -11808.2,E2 -11808.2} C_VEL
LIN {X 0,Y 396.708,Z 175.893,A -85,B 0,C 180,E1 -11808.564,E2 -11808.564} C_VEL
LIN {X 0,Y 395.807,Z 225.253,A -85,B 0,C 180,E1 -11809.496,E2 -11809.496} C_VEL
LIN {X 0,Y 395.2,Z 231.084,A -85,B 0,C 180,E1 -11809.58,E2 -11809.58} C_VEL
LIN {X 0,Y 389.485,Z 250.051,A -85,B 0,C 180,E1 -11809.694,E2 -11809.694} C_VEL
LIN {X 0,Y 388.593,Z 255.875,A -85,B 0,C 180,E1 -11809.784,E2 -11809.784} C_VEL
LIN {X 0,Y 388.228,Z 268.892,A -85,B 0,C 180,E1 -11810.153,E2 -11810.153} C_VEL
LIN {X 0,Y 387.726,Z 281.237,A -85,B 0,C 180,E1 -11810.7,E2 -11810.7} C_VEL
LIN {X 0,Y 387.127,Z 292.726,A -85,B 0,C 180,E1 -11811.401,E2 -11811.401} C_VEL
LIN {X 0,Y 386.478,Z 304.126,A -85,B 0,C 180,E1 -11812.315,E2 -11812.315} C_VEL
LIN {X 0,Y 385.519,Z 315.85,A -85,B 0,C 180,E1 -11813.503,E2 -11813.503} C_VEL
LIN {X 0,Y 384.82,Z 324.896,A -85,B 0,C 180,E1 -11814.646,E2 -11814.646} C_VEL
LIN {X 0,Y 384.071,Z 333.967,A -85,B 0,C 180,E1 -11816.052,E2 -11816.052} C_VEL
LIN {X 0,Y 383.361,Z 341.699,A -85,B 0,C 180,E1 -11817.525,E2 -11817.525} C_VEL
LIN {X 0,Y 382.796,Z 348.438,A -85,B 0,C 180,E1 -11819.114,E2 -11819.114} C_VEL
LIN {X 0,Y 382.313,Z 354.62,A -85,B 0,C 180,E1 -11820.979,E2 -11820.979} C_VEL
LIN {X 0,Y 381.95,Z 359.233,A -85,B 0,C 180,E1 -11822.876,E2 -11822.876} C_VEL
LIN {X 0,Y 381.633,Z 362.468,A -85,B 0,C 180,E1 -11824.813,E2 -11824.813} C_VEL
LIN {X 0,Y 381.507,Z 363.816,A -85,B 0,C 180,E1 -11826.122,E2 -11826.122} C_VEL
LIN {X 0,Y 381.474,Z 364.622,A -85,B 0,C 180,E1 -11827.61,E2 -11827.61} C_VEL
LIN {X 0,Y 381.513,Z 364.556,A -85,B 0,C 180,E1 -11829.314,E2 -11829.314} C_VEL
LIN {X 0,Y 381.653,Z 363.488,A -85,B 0,C 180,E1 -11830.976,E2 -11830.976} C_VEL
LIN {X 0,Y 381.93,Z 360.951,A -85,B 0,C 180,E1 -11832.911,E2 -11832.911} C_VEL
LIN {X 0,Y 382.229,Z 358.201,A -85,B 0,C 180,E1 -11834.324,E2 -11834.324} C_VEL
LIN {X 0,Y 382.641,Z 353.452,A -85,B 0,C 180,E1 -11836.13,E2 -11836.13} C_VEL
LIN {X 0,Y 383.334,Z 347.137,A -85,B 0,C 180,E1 -11837.947,E2 -11837.947} C_VEL
LIN {X 0,Y 384.149,Z 339.521,A -85,B 0,C 180,E1 -11839.639,E2 -11839.639} C_VEL
LIN {X 0,Y 384.989,Z 331.137,A -85,B 0,C 180,E1 -11841.134,E2 -11841.134} C_VEL
LIN {X 0,Y 385.907,Z 322.374,A -85,B 0,C 180,E1 -11842.405,E2 -11842.405} C_VEL
LIN {X 0,Y 386.836,Z 311.684,A -85,B 0,C 180,E1 -11843.659,E2 -11843.659} C_VEL
LIN {X 0,Y 387.915,Z 299.93,A -85,B 0,C 180,E1 -11844.739,E2 -11844.739} C_VEL
LIN {X 0,Y 388.703,Z 287.952,A -85,B 0,C 180,E1 -11845.597,E2 -11845.597} C_VEL
LIN {X 0,Y 389.279,Z 274.776,A -85,B 0,C 180,E1 -11846.288,E2 -11846.288} C_VEL
LIN {X 0,Y 389.734,Z 262.389,A -85,B 0,C 180,E1 -11846.726,E2 -11846.726} C_VEL
LIN {X 0,Y 391.354,Z 176.341,A -85,B 0,C 180,E1 -11848.45,E2 -11848.45} C_VEL
LIN {X 0,Y 388.53,Z 164.012,A -85,B 0,C 180,E1 -11848.892,E2 -11848.892} C_VEL
LIN {X 0,Y 384.987,Z 154.81,A -85,B 0,C 180,E1 -11849.337,E2 -11849.337} C_VEL
LIN {X 0,Y 383.074,Z 145.768,A -85,B 0,C 180,E1 -11851.781,E2 -11851.781} C_VEL
LIN {X 0,Y 383.051,Z 145.776,A -85,B 0,C 180,E1 -11855.04,E2 -11855.04} C_VEL
LIN {X 0,Y 382.995,Z 145.781,A -85,B 0,C 180,E1 -11858.47,E2 -11858.47} C_VEL
LIN {X 0,Y 383.056,Z 145.769,A -85,B 0,C 180,E1 -11861.827,E2 -11861.827} C_VEL
LIN {X 0,Y 383.113,Z 145.767,A -85,B 0,C 180,E1 -11865.119,E2 -11865.119} C_VEL
LIN {X 0,Y 383.101,Z 145.769,A -85,B 0,C 180,E1 -11868.359,E2 -11868.359} C_VEL
LIN {X 0,Y 383.219,Z 145.752,A -85,B 0,C 180,E1 -11872.029,E2 -11872.029} C_VEL
LIN {X 0,Y 383.18,Z 145.755,A -85,B 0,C 180,E1 -11874.739,E2 -11874.739} C_VEL
LIN {X 0,Y 383.378,Z 145.732,A -85,B 0,C 180,E1 -11877.899,E2 -11877.899} C_VEL
LIN {X 0,Y 383.373,Z 145.728,A -85,B 0,C 180,E1 -11882.102,E2 -11882.102} C_VEL
LIN {X 0,Y 383.243,Z 145.739,A -85,B 0,C 180,E1 -11886.318,E2 -11886.318} C_VEL
LIN {X 0,Y 383.14,Z 145.759,A -85,B 0,C 180,E1 -11889.503,E2 -11889.503} C_VEL
LIN {X 0,Y 383.114,Z 145.759,A -85,B 0,C 180,E1 -11892.717,E2 -11892.717} C_VEL
LIN {X 0,Y 383.006,Z 145.772,A -85,B 0,C 180,E1 -11895.977,E2 -11895.977} C_VEL
LIN {X 0,Y 383.004,Z 145.77,A -85,B 0,C 180,E1 -11899.287,E2 -11899.287} C_VEL
LIN {X 0,Y 382.986,Z 145.776,A -85,B 0,C 180,E1 -11902.667,E2 -11902.667} C_VEL
LIN {X 0,Y 382.985,Z 145.777,A -85,B 0,C 180,E1 -11906.131,E2 -11906.131} C_VEL
LIN {X 0,Y 382.978,Z 145.779,A -85,B 0,C 180,E1 -11909.702,E2 -11909.702} C_VEL
LIN {X 0,Y 383.004,Z 145.777,A -85,B 0,C 180,E1 -11913.401,E2 -11913.401} C_VEL
LIN {X 0,Y 383.035,Z 145.77,A -85,B 0,C 180,E1 -11916.164,E2 -11916.164} C_VEL
LIN {X 0,Y 382.98,Z 145.779,A -85,B 0,C 180,E1 -11919.963,E2 -11919.963} C_VEL
LIN {X 0,Y 383.011,Z 145.779,A -85,B 0,C 180,E1 -11922.778,E2 -11922.778} C_VEL
LIN {X 0,Y 383,Z 145.779,A -85,B 0,C 180,E1 -11925.789,E2 -11925.789} C_VEL
LIN {X 0,Y 382.967,Z 145.783,A -85,B 0,C 180,E1 -11928.8,E2 -11928.8} C_VEL
LIN {X 0,Y 382.999,Z 145.779,A -85,B 0,C 180,E1 -11932.097,E2 -11932.097} C_VEL
LIN {X 0,Y 383.023,Z 145.774,A -85,B 0,C 180,E1 -11935.332,E2 -11935.332} C_VEL
LIN {X 0,Y 382.987,Z 145.781,A -85,B 0,C 180,E1 -11939.081,E2 -11939.081} C_VEL
LIN {X 0,Y 383.025,Z 145.874,A -85,B 0,C 180,E1 -11940.037,E2 -11940.037} C_VEL
LIN {X 0,Y 385.734,Z 157.824,A -85,B 0,C 180,E1 -11942.903,E2 -11942.903} C_VEL
LIN {X 0,Y 386.968,Z 164.556,A -85,B 0,C 180,E1 -11944.447,E2 -11944.447} C_VEL
LIN {X 0,Y 386.057,Z 176.674,A -85,B 0,C 180,E1 -11946.958,E2 -11946.958} C_VEL
LIN {X 0,Y 385.356,Z 185.437,A -85,B 0,C 180,E1 -11948.737,E2 -11948.737} C_VEL
LIN {X 0,Y 389.335,Z 208.77,A -85,B 0,C 180,E1 -11949.485,E2 -11949.485} C_VEL
LIN {X 0,Y 390.729,Z 220.252,A -85,B 0,C 180,E1 -11949.81,E2 -11949.81} C_VEL
LIN {X 0,Y 389.375,Z 295.396,A -85,B 0,C 180,E1 -11951.314,E2 -11951.314} C_VEL
LIN {X 0,Y 388.646,Z 308.882,A -85,B 0,C 180,E1 -11951.789,E2 -11951.789} C_VEL
LIN {X 0,Y 387.75,Z 321.692,A -85,B 0,C 180,E1 -11952.462,E2 -11952.462} C_VEL
LIN {X 0,Y 386.766,Z 334.236,A -85,B 0,C 180,E1 -11953.369,E2 -11953.369} C_VEL
LIN {X 0,Y 385.694,Z 345.473,A -85,B 0,C 180,E1 -11954.408,E2 -11954.408} C_VEL
LIN {X 0,Y 384.701,Z 356.407,A -85,B 0,C 180,E1 -11955.694,E2 -11955.694} C_VEL
LIN {X 0,Y 383.856,Z 365.636,A -85,B 0,C 180,E1 -11957.039,E2 -11957.039} C_VEL
LIN {X 0,Y 382.895,Z 374.477,A -85,B 0,C 180,E1 -11958.619,E2 -11958.619} C_VEL
LIN {X 0,Y 382.344,Z 381.55,A -85,B 0,C 180,E1 -11960.21,E2 -11960.21} C_VEL
LIN {X 0,Y 381.896,Z 388.065,A -85,B 0,C 180,E1 -11962.066,E2 -11962.066} C_VEL
LIN {X 0,Y 381.651,Z 393.022,A -85,B 0,C 180,E1 -11963.935,E2 -11963.935} C_VEL
LIN {X 0,Y 381.627,Z 396.437,A -85,B 0,C 180,E1 -11965.775,E2 -11965.775} C_VEL
LIN {X 0,Y 381.655,Z 398.785,A -85,B 0,C 180,E1 -11967.889,E2 -11967.889} C_VEL
LIN {X 0,Y 381.695,Z 399.35,A -85,B 0,C 180,E1 -11968.944,E2 -11968.944} C_VEL
LIN {X 0,Y 381.682,Z 399.47,A -85,B 0,C 180,E1 -11969.999,E2 -11969.999} C_VEL
LIN {X 0,Y 381.695,Z 399.194,A -85,B 0,C 180,E1 -11971.054,E2 -11971.054} C_VEL
LIN {X 0,Y 381.671,Z 398.522,A -85,B 0,C 180,E1 -11972.11,E2 -11972.11} C_VEL
LIN {X 0,Y 381.587,Z 397.431,A -85,B 0,C 180,E1 -11973.167,E2 -11973.167} C_VEL
LIN {X 0,Y 381.633,Z 395.883,A -85,B 0,C 180,E1 -11974.224,E2 -11974.224} C_VEL
LIN {X 0,Y 381.683,Z 392.043,A -85,B 0,C 180,E1 -11976.11,E2 -11976.11} C_VEL
LIN {X 0,Y 381.887,Z 386.888,A -85,B 0,C 180,E1 -11977.933,E2 -11977.933} C_VEL
LIN {X 0,Y 382.28,Z 379.893,A -85,B 0,C 180,E1 -11979.79,E2 -11979.79} C_VEL
LIN {X 0,Y 382.849,Z 372.309,A -85,B 0,C 180,E1 -11981.381,E2 -11981.381} C_VEL
LIN {X 0,Y 383.509,Z 364.566,A -85,B 0,C 180,E1 -11982.703,E2 -11982.703} C_VEL
LIN {X 0,Y 384.315,Z 354.572,A -85,B 0,C 180,E1 -11984.092,E2 -11984.092} C_VEL
LIN {X 0,Y 385.187,Z 343.334,A -85,B 0,C 180,E1 -11985.34,E2 -11985.34} C_VEL
LIN {X 0,Y 386.042,Z 333.005,A -85,B 0,C 180,E1 -11986.254,E2 -11986.254} C_VEL
LIN {X 0,Y 386.914,Z 320.71,A -85,B 0,C 180,E1 -11987.099,E2 -11987.099} C_VEL
LIN {X 0,Y 387.69,Z 307.851,A -85,B 0,C 180,E1 -11987.744,E2 -11987.744} C_VEL
LIN {X 0,Y 388.233,Z 294.312,A -85,B 0,C 180,E1 -11988.195,E2 -11988.195} C_VEL
LIN {X 0,Y 389.333,Z 218.239,A -85,B 0,C 180,E1 -11989.686,E2 -11989.686} C_VEL
LIN {X 0,Y 384.831,Z 186.837,A -85,B 0,C 180,E1 -11990.547,E2 -11990.547} C_VEL
LIN {X 0,Y 386.466,Z 166.541,A -85,B 0,C 180,E1 -11994.724,E2 -11994.724} C_VEL
LIN {X 0,Y 386.462,Z 162.468,A -85,B 0,C 180,E1 -11995.588,E2 -11995.588} C_VEL
LIN {X 0,Y 383.719,Z 148.678,A -85,B 0,C 180,E1 -11998.735,E2 -11998.735} C_VEL
LIN {X 0,Y 383.068,Z 145.769,A -85,B 0,C 180,E1 -11999.466,E2 -11999.466} C_VEL
LIN {X 0,Y 383.013,Z 145.773,A -85,B 0,C 180,E1 -12003.399,E2 -12003.399} C_VEL
LIN {X 0,Y 383.033,Z 145.773,A -85,B 0,C 180,E1 -12006.164,E2 -12006.164} C_VEL
LIN {X 0,Y 383.01,Z 145.778,A -85,B 0,C 180,E1 -12009.958,E2 -12009.958} C_VEL
LIN {X 0,Y 383.005,Z 145.772,A -85,B 0,C 180,E1 -12012.778,E2 -12012.778} C_VEL
LIN {X 0,Y 382.997,Z 145.78,A -85,B 0,C 180,E1 -12015.789,E2 -12015.789} C_VEL
LIN {X 0,Y 382.987,Z 145.775,A -85,B 0,C 180,E1 -12018.795,E2 -12018.795} C_VEL
LIN {X 0,Y 382.997,Z 145.775,A -85,B 0,C 180,E1 -12022.096,E2 -12022.096} C_VEL
LIN {X 0,Y 383.017,Z 145.775,A -85,B 0,C 180,E1 -12025.331,E2 -12025.331} C_VEL
LIN {X 0,Y 382.982,Z 145.778,A -85,B 0,C 180,E1 -12029.081,E2 -12029.081} C_VEL
LIN {X 0,Y 383.056,Z 145.767,A -85,B 0,C 180,E1 -12032.697,E2 -12032.697} C_VEL
LIN {X 0,Y 383.033,Z 145.769,A -85,B 0,C 180,E1 -12036.192,E2 -12036.192} C_VEL
LIN {X 0,Y 383.054,Z 145.769,A -85,B 0,C 180,E1 -12039.598,E2 -12039.598} C_VEL
LIN {X 0,Y 383.092,Z 145.765,A -85,B 0,C 180,E1 -12042.93,E2 -12042.93} C_VEL
LIN {X 0,Y 383.124,Z 145.759,A -85,B 0,C 180,E1 -12046.463,E2 -12046.463} C_VEL
LIN {X 0,Y 383.15,Z 145.756,A -85,B 0,C 180,E1 -12050.497,E2 -12050.497} C_VEL
LIN {X 0,Y 383.278,Z 145.739,A -85,B 0,C 180,E1 -12053.683,E2 -12053.683} C_VEL
LIN {X 0,Y 383.386,Z 145.725,A -85,B 0,C 180,E1 -12057.898,E2 -12057.898} C_VEL
LIN {X 0,Y 383.517,Z 145.709,A -85,B 0,C 180,E1 -12059.999,E2 -12059.999} C_VEL
LIN {X 0,Y 383.248,Z 145.745,A -85,B 0,C 180,E1 -12063.153,E2 -12063.153} C_VEL
LIN {X 0,Y 383.26,Z 145.741,A -85,B 0,C 180,E1 -12066.562,E2 -12066.562} C_VEL
LIN {X 0,Y 383.149,Z 145.755,A -85,B 0,C 180,E1 -12069.502,E2 -12069.502} C_VEL
LIN {X 0,Y 383.122,Z 145.758,A -85,B 0,C 180,E1 -12073.536,E2 -12073.536} C_VEL
LIN {X 0,Y 383.091,Z 145.762,A -85,B 0,C 180,E1 -12077.454,E2 -12077.454} C_VEL
LIN {X 0,Y 383.03,Z 145.773,A -85,B 0,C 180,E1 -12080.649,E2 -12080.649} C_VEL
LIN {X 0,Y 383.029,Z 145.771,A -85,B 0,C 180,E1 -12083.807,E2 -12083.807} C_VEL
LIN {X 0,Y 383.052,Z 145.767,A -85,B 0,C 180,E1 -12087.302,E2 -12087.302} C_VEL
LIN {X 0,Y 382.978,Z 145.776,A -85,B 0,C 180,E1 -12090.918,E2 -12090.918} C_VEL
LIN {X 0,Y 383.013,Z 145.773,A -85,B 0,C 180,E1 -12094.668,E2 -12094.668} C_VEL
LIN {X 0,Y 382.999,Z 145.778,A -85,B 0,C 180,E1 -12097.904,E2 -12097.904} C_VEL
LIN {X 0,Y 383.042,Z 145.769,A -85,B 0,C 180,E1 -12101.339,E2 -12101.339} C_VEL
LIN {X 0,Y 383.066,Z 145.768,A -85,B 0,C 180,E1 -12104.315,E2 -12104.315} C_VEL
LIN {X 0,Y 383.07,Z 145.765,A -85,B 0,C 180,E1 -12107.249,E2 -12107.249} C_VEL
LIN {X 0,Y 383.018,Z 145.772,A -85,B 0,C 180,E1 -12110.412,E2 -12110.412} C_VEL
LIN {X 0,Y 383.022,Z 145.774,A -85,B 0,C 180,E1 -12114.045,E2 -12114.045} C_VEL
LIN {X 0,Y 382.981,Z 145.781,A -85,B 0,C 180,E1 -12117.578,E2 -12117.578} C_VEL
LIN {X 0,Y 382.986,Z 145.775,A -85,B 0,C 180,E1 -12120.3,E2 -12120.3} C_VEL
LIN {X 0,Y 383.051,Z 145.767,A -85,B 0,C 180,E1 -12122.698,E2 -12122.698} C_VEL
LIN {X 0,Y 383.029,Z 145.77,A -85,B 0,C 180,E1 -12126.193,E2 -12126.193} C_VEL
LIN {X 0,Y 383.05,Z 145.772,A -85,B 0,C 180,E1 -12129.599,E2 -12129.599} C_VEL
LIN {X 0,Y 383.1,Z 145.763,A -85,B 0,C 180,E1 -12132.932,E2 -12132.932} C_VEL
LIN {X 0,Y 383.121,Z 145.758,A -85,B 0,C 180,E1 -12136.464,E2 -12136.464} C_VEL
LIN {X 0,Y 383.148,Z 145.755,A -85,B 0,C 180,E1 -12140.498,E2 -12140.498} C_VEL
LIN {X 0,Y 383.269,Z 145.741,A -85,B 0,C 180,E1 -12142.626,E2 -12142.626} C_VEL
LIN {X 0,Y 383.196,Z 145.751,A -85,B 0,C 180,E1 -12144.739,E2 -12144.739} C_VEL
LIN {X 0,Y 383.384,Z 145.725,A -85,B 0,C 180,E1 -12147.9,E2 -12147.9} C_VEL
LIN {X 0,Y 383.516,Z 145.709,A -85,B 0,C 180,E1 -12150.001,E2 -12150.001} C_VEL
LIN {X 0,Y 383.248,Z 145.746,A -85,B 0,C 180,E1 -12153.154,E2 -12153.154} C_VEL
LIN {X 0,Y 383.285,Z 145.739,A -85,B 0,C 180,E1 -12156.317,E2 -12156.317} C_VEL
LIN {X 0,Y 383.257,Z 145.744,A -85,B 0,C 180,E1 -12158.436,E2 -12158.436} C_VEL
LIN {X 0,Y 383.094,Z 145.763,A -85,B 0,C 180,E1 -12161.643,E2 -12161.643} C_VEL
LIN {X 0,Y 383.127,Z 145.764,A -85,B 0,C 180,E1 -12164.882,E2 -12164.882} C_VEL
LIN {X 0,Y 383.182,Z 145.936,A -85,B 0,C 180,E1 -12165.492,E2 -12165.492} C_VEL
LIN {X 0,Y 384.631,Z 153.714,A -85,B 0,C 180,E1 -12167.513,E2 -12167.513} C_VEL
LIN {X 0,Y 387.449,Z 163.332,A -85,B 0,C 180,E1 -12167.859,E2 -12167.859} C_VEL
LIN {X 0,Y 389.956,Z 176.088,A -85,B 0,C 180,E1 -12168.244,E2 -12168.244} C_VEL
LIN {X 0,Y 388.593,Z 255.875,A -85,B 0,C 180,E1 -12169.784,E2 -12169.784} C_VEL
LIN {X 0,Y 387.724,Z 259.783,A -85,B 0,C 180,E1 -12169.837,E2 -12169.837} C_VEL
LIN {X 0,Y 381.786,Z 271.894,A -85,B 0,C 180,E1 -12169.988,E2 -12169.988} C_VEL
LIN {X 0,Y 381.129,Z 275.687,A -85,B 0,C 180,E1 -12170.132,E2 -12170.132} C_VEL
LIN {X 0,Y 380.573,Z 288.374,A -85,B 0,C 180,E1 -12170.824,E2 -12170.824} C_VEL
LIN {X 0,Y 379.889,Z 300.434,A -85,B 0,C 180,E1 -12171.716,E2 -12171.716} C_VEL
LIN {X 0,Y 379.012,Z 311.127,A -85,B 0,C 180,E1 -12172.718,E2 -12172.718} C_VEL
LIN {X 0,Y 378.203,Z 320.798,A -85,B 0,C 180,E1 -12173.84,E2 -12173.84} C_VEL
LIN {X 0,Y 377.472,Z 329.553,A -85,B 0,C 180,E1 -12175.08,E2 -12175.08} C_VEL
LIN {X 0,Y 376.686,Z 338.279,A -85,B 0,C 180,E1 -12176.602,E2 -12176.602} C_VEL
LIN {X 0,Y 376.037,Z 345.605,A -85,B 0,C 180,E1 -12178.182,E2 -12178.182} C_VEL
LIN {X 0,Y 375.433,Z 352.457,A -85,B 0,C 180,E1 -12180.051,E2 -12180.051} C_VEL
LIN {X 0,Y 375.073,Z 356.962,A -85,B 0,C 180,E1 -12181.646,E2 -12181.646} C_VEL
LIN {X 0,Y 374.724,Z 361.001,A -85,B 0,C 180,E1 -12183.593,E2 -12183.593} C_VEL
LIN {X 0,Y 374.451,Z 363.675,A -85,B 0,C 180,E1 -12185.58,E2 -12185.58} C_VEL
LIN {X 0,Y 374.402,Z 364.661,A -85,B 0,C 180,E1 -12186.92,E2 -12186.92} C_VEL
LIN {X 0,Y 374.381,Z 365.061,A -85,B 0,C 180,E1 -12188.28,E2 -12188.28} C_VEL
LIN {X 0,Y 374.448,Z 364.752,A -85,B 0,C 180,E1 -12189.69,E2 -12189.69} C_VEL
LIN {X 0,Y 374.619,Z 363.505,A -85,B 0,C 180,E1 -12191.375,E2 -12191.375} C_VEL
LIN {X 0,Y 374.871,Z 361.32,A -85,B 0,C 180,E1 -12193.017,E2 -12193.017} C_VEL
LIN {X 0,Y 375.21,Z 358.211,A -85,B 0,C 180,E1 -12194.622,E2 -12194.622} C_VEL
LIN {X 0,Y 375.592,Z 354.18,A -85,B 0,C 180,E1 -12196.186,E2 -12196.186} C_VEL
LIN {X 0,Y 376.303,Z 348.148,A -85,B 0,C 180,E1 -12197.986,E2 -12197.986} C_VEL
LIN {X 0,Y 376.996,Z 341.947,A -85,B 0,C 180,E1 -12199.456,E2 -12199.456} C_VEL
LIN {X 0,Y 377.742,Z 335.276,A -85,B 0,C 180,E1 -12200.76,E2 -12200.76} C_VEL
LIN {X 0,Y 378.731,Z 326.069,A -85,B 0,C 180,E1 -12202.24,E2 -12202.24} C_VEL
LIN {X 0,Y 379.638,Z 316.504,A -85,B 0,C 180,E1 -12203.479,E2 -12203.479} C_VEL
LIN {X 0,Y 380.603,Z 306.566,A -85,B 0,C 180,E1 -12204.521,E2 -12204.521} C_VEL
LIN {X 0,Y 381.534,Z 295.278,A -85,B 0,C 180,E1 -12205.47,E2 -12205.47} C_VEL
LIN {X 0,Y 382.31,Z 283.455,A -85,B 0,C 180,E1 -12206.238,E2 -12206.238} C_VEL
LIN {X 0,Y 382.84,Z 271.058,A -85,B 0,C 180,E1 -12206.821,E2 -12206.821} C_VEL
LIN {X 0,Y 383.244,Z 259.265,A -85,B 0,C 180,E1 -12207.185,E2 -12207.185} C_VEL
LIN {X 0,Y 384.902,Z 177.694,A -85,B 0,C 180,E1 -12208.834,E2 -12208.834} C_VEL
LIN {X 0,Y 382.262,Z 166.347,A -85,B 0,C 180,E1 -12209.254,E2 -12209.254} C_VEL
LIN {X 0,Y 377.865,Z 155.17,A -85,B 0,C 180,E1 -12209.818,E2 -12209.818} C_VEL
LIN {X 0,Y 376.035,Z 146.647,A -85,B 0,C 180,E1 -12212.145,E2 -12212.145} C_VEL
LIN {X 0,Y 376.007,Z 146.654,A -85,B 0,C 180,E1 -12214.54,E2 -12214.54} C_VEL
LIN {X 0,Y 375.96,Z 146.657,A -85,B 0,C 180,E1 -12218.046,E2 -12218.046} C_VEL
LIN {X 0,Y 376.006,Z 146.649,A -85,B 0,C 180,E1 -12221.474,E2 -12221.474} C_VEL
LIN {X 0,Y 376.062,Z 146.643,A -85,B 0,C 180,E1 -12224.833,E2 -12224.833} C_VEL
LIN {X 0,Y 376.054,Z 146.646,A -85,B 0,C 180,E1 -12228.137,E2 -12228.137} C_VEL
LIN {X 0,Y 376.191,Z 146.628,A -85,B 0,C 180,E1 -12231.955,E2 -12231.955} C_VEL
LIN {X 0,Y 376.152,Z 146.631,A -85,B 0,C 180,E1 -12234.64,E2 -12234.64} C_VEL
LIN {X 0,Y 376.343,Z 146.608,A -85,B 0,C 180,E1 -12237.86,E2 -12237.86} C_VEL
LIN {X 0,Y 376.337,Z 146.604,A -85,B 0,C 180,E1 -12242.141,E2 -12242.141} C_VEL
LIN {X 0,Y 376.202,Z 146.615,A -85,B 0,C 180,E1 -12246.436,E2 -12246.436} C_VEL
LIN {X 0,Y 376.111,Z 146.635,A -85,B 0,C 180,E1 -12249.682,E2 -12249.682} C_VEL
LIN {X 0,Y 376.045,Z 146.643,A -85,B 0,C 180,E1 -12253.626,E2 -12253.626} C_VEL
LIN {X 0,Y 375.985,Z 146.652,A -85,B 0,C 180,E1 -12257.576,E2 -12257.576} C_VEL
LIN {X 0,Y 375.951,Z 146.651,A -85,B 0,C 180,E1 -12260.819,E2 -12260.819} C_VEL
LIN {X 0,Y 375.936,Z 146.651,A -85,B 0,C 180,E1 -12264.286,E2 -12264.286} C_VEL
LIN {X 0,Y 375.914,Z 146.658,A -85,B 0,C 180,E1 -12266.661,E2 -12266.661} C_VEL
LIN {X 0,Y 375.917,Z 146.658,A -85,B 0,C 180,E1 -12269.084,E2 -12269.084} C_VEL
LIN {X 0,Y 375.941,Z 146.651,A -85,B 0,C 180,E1 -12271.564,E2 -12271.564} C_VEL
LIN {X 0,Y 375.961,Z 146.651,A -85,B 0,C 180,E1 -12275.416,E2 -12275.416} C_VEL
LIN {X 0,Y 375.941,Z 146.652,A -85,B 0,C 180,E1 -12278.263,E2 -12278.263} C_VEL
LIN {X 0,Y 375.922,Z 146.656,A -85,B 0,C 180,E1 -12281.598,E2 -12281.598} C_VEL
LIN {X 0,Y 375.927,Z 146.661,A -85,B 0,C 180,E1 -12284.73,E2 -12284.73} C_VEL
LIN {X 0,Y 375.93,Z 146.66,A -85,B 0,C 180,E1 -12287.699,E2 -12287.699} C_VEL
LIN {X 0,Y 375.94,Z 146.658,A -85,B 0,C 180,E1 -12290.534,E2 -12290.534} C_VEL
LIN {X 0,Y 375.968,Z 146.653,A -85,B 0,C 180,E1 -12293.496,E2 -12293.496} C_VEL
LIN {X 0,Y 375.965,Z 146.657,A -85,B 0,C 180,E1 -12295.888,E2 -12295.888} C_VEL
LIN {X 0,Y 375.974,Z 146.738,A -85,B 0,C 180,E1 -12299.618,E2 -12299.618} C_VEL
LIN {X 0,Y 378.543,Z 157.761,A -85,B 0,C 180,E1 -12302.344,E2 -12302.344} C_VEL
LIN {X 0,Y 380.078,Z 165.828,A -85,B 0,C 180,E1 -12304.243,E2 -12304.243} C_VEL
LIN {X 0,Y 379.378,Z 175.219,A -85,B 0,C 180,E1 -12306.238,E2 -12306.238} C_VEL
LIN {X 0,Y 378.53,Z 184.933,A -85,B 0,C 180,E1 -12308.267,E2 -12308.267} C_VEL
LIN {X 0,Y 382.541,Z 207.796,A -85,B 0,C 180,E1 -12309.037,E2 -12309.037} C_VEL
LIN {X 0,Y 384.181,Z 220.537,A -85,B 0,C 180,E1 -12309.416,E2 -12309.416} C_VEL
LIN {X 0,Y 382.727,Z 295.092,A -85,B 0,C 180,E1 -12310.942,E2 -12310.942} C_VEL
LIN {X 0,Y 381.939,Z 309.286,A -85,B 0,C 180,E1 -12311.458,E2 -12311.458} C_VEL
LIN {X 0,Y 380.991,Z 321.84,A -85,B 0,C 180,E1 -12312.14,E2 -12312.14} C_VEL
LIN {X 0,Y 379.975,Z 334.286,A -85,B 0,C 180,E1 -12313.063,E2 -12313.063} C_VEL
LIN {X 0,Y 378.85,Z 345.452,A -85,B 0,C 180,E1 -12314.119,E2 -12314.119} C_VEL
LIN {X 0,Y 377.844,Z 355.831,A -85,B 0,C 180,E1 -12315.362,E2 -12315.362} C_VEL
LIN {X 0,Y 376.914,Z 365.505,A -85,B 0,C 180,E1 -12316.796,E2 -12316.796} C_VEL
LIN {X 0,Y 375.912,Z 374.305,A -85,B 0,C 180,E1 -12318.405,E2 -12318.405} C_VEL
LIN {X 0,Y 375.301,Z 381.346,A -85,B 0,C 180,E1 -12320.024,E2 -12320.024} C_VEL
LIN {X 0,Y 374.84,Z 387.834,A -85,B 0,C 180,E1 -12321.916,E2 -12321.916} C_VEL
LIN {X 0,Y 374.584,Z 392.102,A -85,B 0,C 180,E1 -12323.536,E2 -12323.536} C_VEL
LIN {X 0,Y 374.529,Z 394.37,A -85,B 0,C 180,E1 -12324.616,E2 -12324.616} C_VEL
LIN {X 0,Y 374.551,Z 396.15,A -85,B 0,C 180,E1 -12325.695,E2 -12325.695} C_VEL
LIN {X 0,Y 374.554,Z 398.48,A -85,B 0,C 180,E1 -12327.849,E2 -12327.849} C_VEL
LIN {X 0,Y 374.626,Z 399.031,A -85,B 0,C 180,E1 -12328.924,E2 -12328.924} C_VEL
LIN {X 0,Y 374.614,Z 399.141,A -85,B 0,C 180,E1 -12329.999,E2 -12329.999} C_VEL
LIN {X 0,Y 374.627,Z 398.857,A -85,B 0,C 180,E1 -12331.074,E2 -12331.074} C_VEL
LIN {X 0,Y 374.571,Z 398.173,A -85,B 0,C 180,E1 -12332.15,E2 -12332.15} C_VEL
LIN {X 0,Y 374.499,Z 397.064,A -85,B 0,C 180,E1 -12333.227,E2 -12333.227} C_VEL
LIN {X 0,Y 374.557,Z 395.505,A -85,B 0,C 180,E1 -12334.304,E2 -12334.304} C_VEL
LIN {X 0,Y 374.58,Z 392.028,A -85,B 0,C 180,E1 -12336.059,E2 -12336.059} C_VEL
LIN {X 0,Y 374.83,Z 386.454,A -85,B 0,C 180,E1 -12338.083,E2 -12338.083} C_VEL
LIN {X 0,Y 375.25,Z 379.423,A -85,B 0,C 180,E1 -12339.976,E2 -12339.976} C_VEL
LIN {X 0,Y 375.859,Z 371.806,A -85,B 0,C 180,E1 -12341.595,E2 -12341.595} C_VEL
LIN {X 0,Y 376.51,Z 364.02,A -85,B 0,C 180,E1 -12342.943,E2 -12342.943} C_VEL
LIN {X 0,Y 377.301,Z 354.958,A -85,B 0,C 180,E1 -12344.232,E2 -12344.232} C_VEL
LIN {X 0,Y 378.189,Z 343.95,A -85,B 0,C 180,E1 -12345.493,E2 -12345.493} C_VEL
LIN {X 0,Y 379.213,Z 332.23,A -85,B 0,C 180,E1 -12346.555,E2 -12346.555} C_VEL
LIN {X 0,Y 380.114,Z 319.741,A -85,B 0,C 180,E1 -12347.415,E2 -12347.415} C_VEL
LIN {X 0,Y 380.917,Z 306.66,A -85,B 0,C 180,E1 -12348.07,E2 -12348.07} C_VEL
LIN {X 0,Y 381.415,Z 293.756,A -85,B 0,C 180,E1 -12348.498,E2 -12348.498} C_VEL
LIN {X 0,Y 382.554,Z 218.865,A -85,B 0,C 180,E1 -12349.993,E2 -12349.993} C_VEL
LIN {X 0,Y 377.926,Z 186.541,A -85,B 0,C 180,E1 -12350.9,E2 -12350.9} C_VEL
LIN {X 0,Y 379.52,Z 167.665,A -85,B 0,C 180,E1 -12354.852,E2 -12354.852} C_VEL
LIN {X 0,Y 379.423,Z 163.299,A -85,B 0,C 180,E1 -12355.803,E2 -12355.803} C_VEL
LIN {X 0,Y 376.88,Z 150.482,A -85,B 0,C 180,E1 -12358.782,E2 -12358.782} C_VEL
LIN {X 0,Y 376.011,Z 146.649,A -85,B 0,C 180,E1 -12359.728,E2 -12359.728} C_VEL
LIN {X 0,Y 375.952,Z 146.654,A -85,B 0,C 180,E1 -12362.828,E2 -12362.828} C_VEL
LIN {X 0,Y 375.958,Z 146.652,A -85,B 0,C 180,E1 -12365.415,E2 -12365.415} C_VEL
LIN {X 0,Y 375.975,Z 146.651,A -85,B 0,C 180,E1 -12368.27,E2 -12368.27} C_VEL
LIN {X 0,Y 375.935,Z 146.657,A -85,B 0,C 180,E1 -12371.6,E2 -12371.6} C_VEL
LIN {X 0,Y 375.927,Z 146.656,A -85,B 0,C 180,E1 -12375.268,E2 -12375.268} C_VEL
LIN {X 0,Y 375.934,Z 146.654,A -85,B 0,C 180,E1 -12378.399,E2 -12378.399} C_VEL
LIN {X 0,Y 375.972,Z 146.654,A -85,B 0,C 180,E1 -12381.729,E2 -12381.729} C_VEL
LIN {X 0,Y 375.979,Z 146.652,A -85,B 0,C 180,E1 -12385.332,E2 -12385.332} C_VEL
LIN {X 0,Y 375.956,Z 146.651,A -85,B 0,C 180,E1 -12388.437,E2 -12388.437} C_VEL
LIN {X 0,Y 375.995,Z 146.646,A -85,B 0,C 180,E1 -12392.141,E2 -12392.141} C_VEL
LIN {X 0,Y 376.005,Z 146.645,A -85,B 0,C 180,E1 -12394.538,E2 -12394.538} C_VEL
LIN {X 0,Y 375.962,Z 146.65,A -85,B 0,C 180,E1 -12398.045,E2 -12398.045} C_VEL
LIN {X 0,Y 376.001,Z 146.649,A -85,B 0,C 180,E1 -12401.472,E2 -12401.472} C_VEL
LIN {X 0,Y 376.057,Z 146.641,A -85,B 0,C 180,E1 -12404.832,E2 -12404.832} C_VEL
LIN {X 0,Y 376.048,Z 146.639,A -85,B 0,C 180,E1 -12408.136,E2 -12408.136} C_VEL
LIN {X 0,Y 376.217,Z 146.618,A -85,B 0,C 180,E1 -12411.918,E2 -12411.918} C_VEL
LIN {X 0,Y 376.168,Z 146.627,A -85,B 0,C 180,E1 -12414.639,E2 -12414.639} C_VEL
LIN {X 0,Y 376.352,Z 146.601,A -85,B 0,C 180,E1 -12417.859,E2 -12417.859} C_VEL
LIN {X 0,Y 376.487,Z 146.585,A -85,B 0,C 180,E1 -12419.999,E2 -12419.999} C_VEL
LIN {X 0,Y 376.186,Z 146.624,A -85,B 0,C 180,E1 -12423.212,E2 -12423.212} C_VEL
LIN {X 0,Y 376.226,Z 146.619,A -85,B 0,C 180,E1 -12426.549,E2 -12426.549} C_VEL
LIN {X 0,Y 376.116,Z 146.631,A -85,B 0,C 180,E1 -12429.681,E2 -12429.681} C_VEL
LIN {X 0,Y 376.086,Z 146.635,A -85,B 0,C 180,E1 -12433.657,E2 -12433.657} C_VEL
LIN {X 0,Y 376.04,Z 146.64,A -85,B 0,C 180,E1 -12437.607,E2 -12437.607} C_VEL
LIN {X 0,Y 375.974,Z 146.651,A -85,B 0,C 180,E1 -12440.832,E2 -12440.832} C_VEL
LIN {X 0,Y 375.99,Z 146.652,A -85,B 0,C 180,E1 -12444.281,E2 -12444.281} C_VEL
LIN {X 0,Y 376.015,Z 146.646,A -85,B 0,C 180,E1 -12446.652,E2 -12446.652} C_VEL
LIN {X 0,Y 375.966,Z 146.65,A -85,B 0,C 180,E1 -12449.079,E2 -12449.079} C_VEL
LIN {X 0,Y 375.946,Z 146.653,A -85,B 0,C 180,E1 -12452.828,E2 -12452.828} C_VEL
LIN {X 0,Y 375.954,Z 146.652,A -85,B 0,C 180,E1 -12455.415,E2 -12455.415} C_VEL
LIN {X 0,Y 375.973,Z 146.653,A -85,B 0,C 180,E1 -12458.271,E2 -12458.271} C_VEL
LIN {X 0,Y 375.985,Z 146.65,A -85,B 0,C 180,E1 -12461.61,E2 -12461.61} C_VEL
LIN {X 0,Y 376.012,Z 146.644,A -85,B 0,C 180,E1 -12465.255,E2 -12465.255} C_VEL
LIN {X 0,Y 375.985,Z 146.649,A -85,B 0,C 180,E1 -12468.39,E2 -12468.39} C_VEL
LIN {X 0,Y 375.963,Z 146.655,A -85,B 0,C 180,E1 -12471.912,E2 -12471.912} C_VEL
LIN {X 0,Y 375.975,Z 146.651,A -85,B 0,C 180,E1 -12475.333,E2 -12475.333} C_VEL
LIN {X 0,Y 375.952,Z 146.651,A -85,B 0,C 180,E1 -12478.438,E2 -12478.438} C_VEL
LIN {X 0,Y 375.991,Z 146.648,A -85,B 0,C 180,E1 -12482.142,E2 -12482.142} C_VEL
LIN {X 0,Y 376.001,Z 146.645,A -85,B 0,C 180,E1 -12484.539,E2 -12484.539} C_VEL
LIN {X 0,Y 375.958,Z 146.651,A -85,B 0,C 180,E1 -12488.046,E2 -12488.046} C_VEL
LIN {X 0,Y 376.019,Z 146.648,A -85,B 0,C 180,E1 -12491.474,E2 -12491.474} C_VEL
LIN {X 0,Y 376.054,Z 146.64,A -85,B 0,C 180,E1 -12494.833,E2 -12494.833} C_VEL
LIN {X 0,Y 376.046,Z 146.64,A -85,B 0,C 180,E1 -12498.137,E2 -12498.137} C_VEL
LIN {X 0,Y 376.253,Z 146.614,A -85,B 0,C 180,E1 -12501.878,E2 -12501.878} C_VEL
LIN {X 0,Y 376.169,Z 146.626,A -85,B 0,C 180,E1 -12504.64,E2 -12504.64} C_VEL
LIN {X 0,Y 376.35,Z 146.602,A -85,B 0,C 180,E1 -12507.86,E2 -12507.86} C_VEL
LIN {X 0,Y 376.486,Z 146.585,A -85,B 0,C 180,E1 -12510.001,E2 -12510.001} C_VEL
LIN {X 0,Y 376.186,Z 146.625,A -85,B 0,C 180,E1 -12513.214,E2 -12513.214} C_VEL
LIN {X 0,Y 376.244,Z 146.617,A -85,B 0,C 180,E1 -12516.436,E2 -12516.436} C_VEL
LIN {X 0,Y 376.202,Z 146.624,A -85,B 0,C 180,E1 -12518.596,E2 -12518.596} C_VEL
LIN {X 0,Y 376.045,Z 146.641,A -85,B 0,C 180,E1 -12521.864,E2 -12521.864} C_VEL
LIN {X 0,Y 376.113,Z 146.773,A -85,B 0,C 180,E1 -12525.235,E2 -12525.235} C_VEL
LIN {X 0,Y 377.476,Z 154.043,A -85,B 0,C 180,E1 -12527.157,E2 -12527.157} C_VEL
LIN {X 0,Y 380.795,Z 164.784,A -85,B 0,C 180,E1 -12527.557,E2 -12527.557} C_VEL
LIN {X 0,Y 383.185,Z 176.775,A -85,B 0,C 180,E1 -12527.926,E2 -12527.926} C_VEL
LIN {X 0,Y 381.615,Z 261.929,A -85,B 0,C 180,E1 -12529.628,E2 -12529.628} C_VEL
LIN {X 0,Y 381.129,Z 275.687,A -85,B 0,C 180,E1 -12530.132,E2 -12530.132} C_VEL
LIN {X 0,Y 380.428,Z 279.474,A -85,B 0,C 180,E1 -12530.285,E2 -12530.285} C_VEL
LIN {X 0,Y 377.385,Z 285.376,A -85,B 0,C 180,E1 -12530.483,E2 -12530.483} C_VEL
LIN {X 0,Y 374.221,Z 291.146,A -85,B 0,C 180,E1 -12530.734,E2 -12530.734} C_VEL
LIN {X 0,Y 373.337,Z 294.728,A -85,B 0,C 180,E1 -12530.969,E2 -12530.969} C_VEL
LIN {X 0,Y 372.491,Z 307.037,A -85,B 0,C 180,E1 -12532.025,E2 -12532.025} C_VEL
LIN {X 0,Y 371.64,Z 317.111,A -85,B 0,C 180,E1 -12533.113,E2 -12533.113} C_VEL
LIN {X 0,Y 370.752,Z 327.453,A -85,B 0,C 180,E1 -12534.512,E2 -12534.512} C_VEL
LIN {X 0,Y 369.865,Z 336.885,A -85,B 0,C 180,E1 -12536.096,E2 -12536.096} C_VEL
LIN {X 0,Y 369.201,Z 343.635,A -85,B 0,C 180,E1 -12537.492,E2 -12537.492} C_VEL
LIN {X 0,Y 368.595,Z 350.343,A -85,B 0,C 180,E1 -12539.205,E2 -12539.205} C_VEL
LIN {X 0,Y 368.137,Z 355.89,A -85,B 0,C 180,E1 -12541.028,E2 -12541.028} C_VEL
LIN {X 0,Y 367.783,Z 359.917,A -85,B 0,C 180,E1 -12542.777,E2 -12542.777} C_VEL
LIN {X 0,Y 367.468,Z 362.993,A -85,B 0,C 180,E1 -12544.676,E2 -12544.676} C_VEL
LIN {X 0,Y 367.319,Z 364.772,A -85,B 0,C 180,E1 -12546.526,E2 -12546.526} C_VEL
LIN {X 0,Y 367.288,Z 365.389,A -85,B 0,C 180,E1 -12548.324,E2 -12548.324} C_VEL
LIN {X 0,Y 367.382,Z 364.95,A -85,B 0,C 180,E1 -12550.077,E2 -12550.077} C_VEL
LIN {X 0,Y 367.619,Z 363.273,A -85,B 0,C 180,E1 -12552,E2 -12552} C_VEL
LIN {X 0,Y 367.88,Z 361.168,A -85,B 0,C 180,E1 -12553.453,E2 -12553.453} C_VEL
LIN {X 0,Y 368.225,Z 357.9,A -85,B 0,C 180,E1 -12555.075,E2 -12555.075} C_VEL
LIN {X 0,Y 368.689,Z 353.671,A -85,B 0,C 180,E1 -12556.668,E2 -12556.668} C_VEL
LIN {X 0,Y 369.446,Z 347.48,A -85,B 0,C 180,E1 -12558.481,E2 -12558.481} C_VEL
LIN {X 0,Y 370.278,Z 340.378,A -85,B 0,C 180,E1 -12560.113,E2 -12560.113} C_VEL
LIN {X 0,Y 371.336,Z 331.19,A -85,B 0,C 180,E1 -12561.806,E2 -12561.806} C_VEL
LIN {X 0,Y 372.417,Z 321.928,A -85,B 0,C 180,E1 -12563.167,E2 -12563.167} C_VEL
LIN {X 0,Y 373.329,Z 312.522,A -85,B 0,C 180,E1 -12564.298,E2 -12564.298} C_VEL
LIN {X 0,Y 374.481,Z 301.115,A -85,B 0,C 180,E1 -12565.39,E2 -12565.39} C_VEL
LIN {X 0,Y 375.275,Z 290.135,A -85,B 0,C 180,E1 -12566.223,E2 -12566.223} C_VEL
LIN {X 0,Y 375.924,Z 277.411,A -85,B 0,C 180,E1 -12566.95,E2 -12566.95} C_VEL
LIN {X 0,Y 376.493,Z 263.975,A -85,B 0,C 180,E1 -12567.464,E2 -12567.464} C_VEL
LIN {X 0,Y 377.357,Z 224.054,A -85,B 0,C 180,E1 -12568.315,E2 -12568.315} C_VEL
LIN {X 0,Y 378.387,Z 178.713,A -85,B 0,C 180,E1 -12569.242,E2 -12569.242} C_VEL
LIN {X 0,Y 375.909,Z 168.354,A -85,B 0,C 180,E1 -12569.644,E2 -12569.644} C_VEL
LIN {X 0,Y 370.777,Z 155.511,A -85,B 0,C 180,E1 -12570.334,E2 -12570.334} C_VEL
LIN {X 0,Y 368.975,Z 147.527,A -85,B 0,C 180,E1 -12572.568,E2 -12572.568} C_VEL
LIN {X 0,Y 368.956,Z 147.533,A -85,B 0,C 180,E1 -12575.225,E2 -12575.225} C_VEL
LIN {X 0,Y 368.923,Z 147.533,A -85,B 0,C 180,E1 -12578.982,E2 -12578.982} C_VEL
LIN {X 0,Y 368.994,Z 147.521,A -85,B 0,C 180,E1 -12582.258,E2 -12582.258} C_VEL
LIN {X 0,Y 369.041,Z 147.519,A -85,B 0,C 180,E1 -12586.229,E2 -12586.229} C_VEL
LIN {X 0,Y 369.067,Z 147.512,A -85,B 0,C 180,E1 -12590.132,E2 -12590.132} C_VEL
LIN {X 0,Y 369.163,Z 147.501,A -85,B 0,C 180,E1 -12593.442,E2 -12593.442} C_VEL
LIN {X 0,Y 369.307,Z 147.484,A -85,B 0,C 180,E1 -12597.819,E2 -12597.819} C_VEL
LIN {X 0,Y 369.3,Z 147.479,A -85,B 0,C 180,E1 -12602.182,E2 -12602.182} C_VEL
LIN {X 0,Y 369.164,Z 147.49,A -85,B 0,C 180,E1 -12606.56,E2 -12606.56} C_VEL
LIN {X 0,Y 369.061,Z 147.51,A -85,B 0,C 180,E1 -12609.869,E2 -12609.869} C_VEL
LIN {X 0,Y 369.006,Z 147.518,A -85,B 0,C 180,E1 -12613.749,E2 -12613.749} C_VEL
LIN {X 0,Y 368.941,Z 147.527,A -85,B 0,C 180,E1 -12617.746,E2 -12617.746} C_VEL
LIN {X 0,Y 368.884,Z 147.535,A -85,B 0,C 180,E1 -12621.223,E2 -12621.223} C_VEL
LIN {X 0,Y 368.91,Z 147.525,A -85,B 0,C 180,E1 -12623.873,E2 -12623.873} C_VEL
LIN {X 0,Y 368.861,Z 147.533,A -85,B 0,C 180,E1 -12627.212,E2 -12627.212} C_VEL
LIN {X 0,Y 368.896,Z 147.533,A -85,B 0,C 180,E1 -12629.693,E2 -12629.693} C_VEL
LIN {X 0,Y 368.901,Z 147.534,A -85,B 0,C 180,E1 -12633.043,E2 -12633.043} C_VEL
LIN {X 0,Y 368.921,Z 147.528,A -85,B 0,C 180,E1 -12636.197,E2 -12636.197} C_VEL
LIN {X 0,Y 368.879,Z 147.534,A -85,B 0,C 180,E1 -12638.957,E2 -12638.957} C_VEL
LIN {X 0,Y 368.875,Z 147.535,A -85,B 0,C 180,E1 -12642.007,E2 -12642.007} C_VEL
LIN {X 0,Y 368.882,Z 147.539,A -85,B 0,C 180,E1 -12645.175,E2 -12645.175} C_VEL
LIN {X 0,Y 368.875,Z 147.541,A -85,B 0,C 180,E1 -12648.176,E2 -12648.176} C_VEL
LIN {X 0,Y 368.882,Z 147.536,A -85,B 0,C 180,E1 -12651.366,E2 -12651.366} C_VEL
LIN {X 0,Y 368.942,Z 147.529,A -85,B 0,C 180,E1 -12655.146,E2 -12655.146} C_VEL
LIN {X 0,Y 368.922,Z 147.539,A -85,B 0,C 180,E1 -12659.164,E2 -12659.164} C_VEL
LIN {X 0,Y 371.792,Z 159.873,A -85,B 0,C 180,E1 -12662.293,E2 -12662.293} C_VEL
LIN {X 0,Y 373.174,Z 167.111,A -85,B 0,C 180,E1 -12664.031,E2 -12664.031} C_VEL
LIN {X 0,Y 372.626,Z 175.157,A -85,B 0,C 180,E1 -12665.781,E2 -12665.781} C_VEL
LIN {X 0,Y 371.705,Z 184.538,A -85,B 0,C 180,E1 -12667.78,E2 -12667.78} C_VEL
LIN {X 0,Y 375.263,Z 203.976,A -85,B 0,C 180,E1 -12668.478,E2 -12668.478} C_VEL
LIN {X 0,Y 377.603,Z 221.758,A -85,B 0,C 180,E1 -12669.024,E2 -12669.024} C_VEL
LIN {X 0,Y 376.147,Z 293.981,A -85,B 0,C 180,E1 -12670.524,E2 -12670.524} C_VEL
LIN {X 0,Y 375.402,Z 307.65,A -85,B 0,C 180,E1 -12671.017,E2 -12671.017} C_VEL
LIN {X 0,Y 374.5,Z 320.072,A -85,B 0,C 180,E1 -12671.679,E2 -12671.679} C_VEL
LIN {X 0,Y 373.478,Z 331.238,A -85,B 0,C 180,E1 -12672.477,E2 -12672.477} C_VEL
LIN {X 0,Y 372.275,Z 342.873,A -85,B 0,C 180,E1 -12673.549,E2 -12673.549} C_VEL
LIN {X 0,Y 371.12,Z 354.013,A -85,B 0,C 180,E1 -12674.848,E2 -12674.848} C_VEL
LIN {X 0,Y 370.11,Z 363.723,A -85,B 0,C 180,E1 -12676.268,E2 -12676.268} C_VEL
LIN {X 0,Y 369.117,Z 372.786,A -85,B 0,C 180,E1 -12677.91,E2 -12677.91} C_VEL
LIN {X 0,Y 368.387,Z 380.101,A -85,B 0,C 180,E1 -12679.557,E2 -12679.557} C_VEL
LIN {X 0,Y 367.883,Z 385.952,A -85,B 0,C 180,E1 -12681.208,E2 -12681.208} C_VEL
LIN {X 0,Y 367.596,Z 390.576,A -85,B 0,C 180,E1 -12682.861,E2 -12682.861} C_VEL
LIN {X 0,Y 367.446,Z 394.104,A -85,B 0,C 180,E1 -12684.512,E2 -12684.512} C_VEL
LIN {X 0,Y 367.454,Z 395.87,A -85,B 0,C 180,E1 -12685.612,E2 -12685.612} C_VEL
LIN {X 0,Y 367.453,Z 398.181,A -85,B 0,C 180,E1 -12687.807,E2 -12687.807} C_VEL
LIN {X 0,Y 367.54,Z 398.71,A -85,B 0,C 180,E1 -12688.904,E2 -12688.904} C_VEL
LIN {X 0,Y 367.547,Z 398.81,A -85,B 0,C 180,E1 -12689.999,E2 -12689.999} C_VEL
LIN {X 0,Y 367.542,Z 398.515,A -85,B 0,C 180,E1 -12691.095,E2 -12691.095} C_VEL
LIN {X 0,Y 367.471,Z 397.82,A -85,B 0,C 180,E1 -12692.192,E2 -12692.192} C_VEL
LIN {X 0,Y 367.414,Z 396.689,A -85,B 0,C 180,E1 -12693.289,E2 -12693.289} C_VEL
LIN {X 0,Y 367.437,Z 394.193,A -85,B 0,C 180,E1 -12694.937,E2 -12694.937} C_VEL
LIN {X 0,Y 367.555,Z 390.66,A -85,B 0,C 180,E1 -12696.587,E2 -12696.587} C_VEL
LIN {X 0,Y 367.766,Z 385.996,A -85,B 0,C 180,E1 -12698.24,E2 -12698.24} C_VEL
LIN {X 0,Y 368.225,Z 378.925,A -85,B 0,C 180,E1 -12700.168,E2 -12700.168} C_VEL
LIN {X 0,Y 368.868,Z 371.263,A -85,B 0,C 180,E1 -12701.818,E2 -12701.818} C_VEL
LIN {X 0,Y 369.535,Z 363.416,A -85,B 0,C 180,E1 -12703.192,E2 -12703.192} C_VEL
LIN {X 0,Y 370.393,Z 353.506,A -85,B 0,C 180,E1 -12704.601,E2 -12704.601} C_VEL
LIN {X 0,Y 371.339,Z 343.187,A -85,B 0,C 180,E1 -12705.786,E2 -12705.786} C_VEL
LIN {X 0,Y 372.371,Z 331.327,A -85,B 0,C 180,E1 -12706.868,E2 -12706.868} C_VEL
LIN {X 0,Y 373.301,Z 318.643,A -85,B 0,C 180,E1 -12707.743,E2 -12707.743} C_VEL
LIN {X 0,Y 374.087,Z 306.057,A -85,B 0,C 180,E1 -12708.376,E2 -12708.376} C_VEL
LIN {X 0,Y 374.627,Z 292.907,A -85,B 0,C 180,E1 -12708.81,E2 -12708.81} C_VEL
LIN {X 0,Y 375.819,Z 219.869,A -85,B 0,C 180,E1 -12710.294,E2 -12710.294} C_VEL
LIN {X 0,Y 371.011,Z 186.254,A -85,B 0,C 180,E1 -12711.256,E2 -12711.256} C_VEL
LIN {X 0,Y 372.635,Z 168.095,A -85,B 0,C 180,E1 -12715.136,E2 -12715.136} C_VEL
LIN {X 0,Y 372.373,Z 164.124,A -85,B 0,C 180,E1 -12716.027,E2 -12716.027} C_VEL
LIN {X 0,Y 370,Z 152.161,A -85,B 0,C 180,E1 -12718.86,E2 -12718.86} C_VEL
LIN {X 0,Y 368.953,Z 147.529,A -85,B 0,C 180,E1 -12720.001,E2 -12720.001} C_VEL
LIN {X 0,Y 368.899,Z 147.532,A -85,B 0,C 180,E1 -12723.537,E2 -12723.537} C_VEL
LIN {X 0,Y 368.902,Z 147.529,A -85,B 0,C 180,E1 -12726.855,E2 -12726.855} C_VEL
LIN {X 0,Y 368.911,Z 147.53,A -85,B 0,C 180,E1 -12730.369,E2 -12730.369} C_VEL
LIN {X 0,Y 368.883,Z 147.536,A -85,B 0,C 180,E1 -12733.615,E2 -12733.615} C_VEL
LIN {X 0,Y 368.885,Z 147.532,A -85,B 0,C 180,E1 -12736.695,E2 -12736.695} C_VEL
LIN {X 0,Y 368.911,Z 147.535,A -85,B 0,C 180,E1 -12739.642,E2 -12739.642} C_VEL
LIN {X 0,Y 368.9,Z 147.532,A -85,B 0,C 180,E1 -12743.144,E2 -12743.144} C_VEL
LIN {X 0,Y 368.895,Z 147.53,A -85,B 0,C 180,E1 -12746.461,E2 -12746.461} C_VEL
LIN {X 0,Y 368.928,Z 147.528,A -85,B 0,C 180,E1 -12749.046,E2 -12749.046} C_VEL
LIN {X 0,Y 368.979,Z 147.525,A -85,B 0,C 180,E1 -12751.563,E2 -12751.563} C_VEL
LIN {X 0,Y 368.999,Z 147.518,A -85,B 0,C 180,E1 -12754.019,E2 -12754.019} C_VEL
LIN {X 0,Y 368.931,Z 147.529,A -85,B 0,C 180,E1 -12757.604,E2 -12757.604} C_VEL
LIN {X 0,Y 368.952,Z 147.528,A -85,B 0,C 180,E1 -12761.105,E2 -12761.105} C_VEL
LIN {X 0,Y 368.995,Z 147.519,A -85,B 0,C 180,E1 -12764.534,E2 -12764.534} C_VEL
LIN {X 0,Y 369.003,Z 147.517,A -85,B 0,C 180,E1 -12767.906,E2 -12767.906} C_VEL
LIN {X 0,Y 369.185,Z 147.494,A -85,B 0,C 180,E1 -12771.845,E2 -12771.845} C_VEL
LIN {X 0,Y 369.14,Z 147.502,A -85,B 0,C 180,E1 -12774.537,E2 -12774.537} C_VEL
LIN {X 0,Y 369.317,Z 147.478,A -85,B 0,C 180,E1 -12777.818,E2 -12777.818} C_VEL
LIN {X 0,Y 369.456,Z 147.46,A -85,B 0,C 180,E1 -12779.999,E2 -12779.999} C_VEL
LIN {X 0,Y 369.316,Z 147.479,A -85,B 0,C 180,E1 -12782.181,E2 -12782.181} C_VEL
LIN {X 0,Y 369.196,Z 147.498,A -85,B 0,C 180,E1 -12786.558,E2 -12786.558} C_VEL
LIN {X 0,Y 369.118,Z 147.508,A -85,B 0,C 180,E1 -12788.761,E2 -12788.761} C_VEL
LIN {X 0,Y 369.002,Z 147.519,A -85,B 0,C 180,E1 -12792.093,E2 -12792.093} C_VEL
LIN {X 0,Y 368.995,Z 147.518,A -85,B 0,C 180,E1 -12795.464,E2 -12795.464} C_VEL
LIN {X 0,Y 368.98,Z 147.522,A -85,B 0,C 180,E1 -12798.892,E2 -12798.892} C_VEL
LIN {X 0,Y 368.929,Z 147.533,A -85,B 0,C 180,E1 -12802.395,E2 -12802.395} C_VEL
LIN {X 0,Y 368.996,Z 147.521,A -85,B 0,C 180,E1 -12805.98,E2 -12805.98} C_VEL
LIN {X 0,Y 368.957,Z 147.524,A -85,B 0,C 180,E1 -12808.811,E2 -12808.811} C_VEL
LIN {X 0,Y 368.894,Z 147.536,A -85,B 0,C 180,E1 -12812.238,E2 -12812.238} C_VEL
LIN {X 0,Y 368.925,Z 147.527,A -85,B 0,C 180,E1 -12815.001,E2 -12815.001} C_VEL
LIN {X 0,Y 368.909,Z 147.53,A -85,B 0,C 180,E1 -12818.641,E2 -12818.641} C_VEL
LIN {X 0,Y 368.947,Z 147.53,A -85,B 0,C 180,E1 -12822.022,E2 -12822.022} C_VEL
LIN {X 0,Y 368.986,Z 147.519,A -85,B 0,C 180,E1 -12825.193,E2 -12825.193} C_VEL
LIN {X 0,Y 368.941,Z 147.528,A -85,B 0,C 180,E1 -12828.186,E2 -12828.186} C_VEL
LIN {X 0,Y 368.908,Z 147.531,A -85,B 0,C 180,E1 -12831.359,E2 -12831.359} C_VEL
LIN {X 0,Y 368.932,Z 147.527,A -85,B 0,C 180,E1 -12835.147,E2 -12835.147} C_VEL
LIN {X 0,Y 368.924,Z 147.528,A -85,B 0,C 180,E1 -12839.047,E2 -12839.047} C_VEL
LIN {X 0,Y 368.974,Z 147.527,A -85,B 0,C 180,E1 -12841.564,E2 -12841.564} C_VEL
LIN {X 0,Y 368.995,Z 147.52,A -85,B 0,C 180,E1 -12844.02,E2 -12844.02} C_VEL
LIN {X 0,Y 368.928,Z 147.531,A -85,B 0,C 180,E1 -12847.605,E2 -12847.605} C_VEL
LIN {X 0,Y 368.978,Z 147.523,A -85,B 0,C 180,E1 -12851.108,E2 -12851.108} C_VEL
LIN {X 0,Y 368.993,Z 147.518,A -85,B 0,C 180,E1 -12854.536,E2 -12854.536} C_VEL
LIN {X 0,Y 369.001,Z 147.518,A -85,B 0,C 180,E1 -12857.907,E2 -12857.907} C_VEL
LIN {X 0,Y 369.225,Z 147.49,A -85,B 0,C 180,E1 -12861.801,E2 -12861.801} C_VEL
LIN {X 0,Y 369.142,Z 147.501,A -85,B 0,C 180,E1 -12864.538,E2 -12864.538} C_VEL
LIN {X 0,Y 369.315,Z 147.478,A -85,B 0,C 180,E1 -12867.819,E2 -12867.819} C_VEL
LIN {X 0,Y 369.455,Z 147.46,A -85,B 0,C 180,E1 -12870.001,E2 -12870.001} C_VEL
LIN {X 0,Y 369.316,Z 147.478,A -85,B 0,C 180,E1 -12872.182,E2 -12872.182} C_VEL
LIN {X 0,Y 369.206,Z 147.495,A -85,B 0,C 180,E1 -12876.559,E2 -12876.559} C_VEL
LIN {X 0,Y 369.135,Z 147.506,A -85,B 0,C 180,E1 -12878.762,E2 -12878.762} C_VEL
LIN {X 0,Y 368.999,Z 147.519,A -85,B 0,C 180,E1 -12882.094,E2 -12882.094} C_VEL
LIN {X 0,Y 369.076,Z 147.605,A -85,B 0,C 180,E1 -12884.967,E2 -12884.967} C_VEL
LIN {X 0,Y 370.365,Z 154.385,A -85,B 0,C 180,E1 -12886.786,E2 -12886.786} C_VEL
LIN {X 0,Y 374.156,Z 166.209,A -85,B 0,C 180,E1 -12887.244,E2 -12887.244} C_VEL
LIN {X 0,Y 376.455,Z 177.797,A -85,B 0,C 180,E1 -12887.609,E2 -12887.609} C_VEL
LIN {X 0,Y 374.803,Z 262.429,A -85,B 0,C 180,E1 -12889.335,E2 -12889.335} C_VEL
LIN {X 0,Y 374.304,Z 276.228,A -85,B 0,C 180,E1 -12889.852,E2 -12889.852} C_VEL
LIN {X 0,Y 373.707,Z 289.07,A -85,B 0,C 180,E1 -12890.572,E2 -12890.572} C_VEL
LIN {X 0,Y 373.337,Z 294.728,A -85,B 0,C 180,E1 -12890.969,E2 -12890.969} C_VEL
LIN {X 0,Y 372.374,Z 300.064,A -85,B 0,C 180,E1 -12891.365,E2 -12891.365} C_VEL
LIN {X 0,Y 368.953,Z 308.412,A -85,B 0,C 180,E1 -12892.014,E2 -12892.014} C_VEL
LIN {X 0,Y 365.467,Z 316.295,A -85,B 0,C 180,E1 -12892.764,E2 -12892.764} C_VEL
LIN {X 0,Y 364.402,Z 320.864,A -85,B 0,C 180,E1 -12893.312,E2 -12893.312} C_VEL
LIN {X 0,Y 363.544,Z 330.303,A -85,B 0,C 180,E1 -12894.689,E2 -12894.689} C_VEL
LIN {X 0,Y 362.743,Z 338.45,A -85,B 0,C 180,E1 -12896.154,E2 -12896.154} C_VEL
LIN {X 0,Y 362.038,Z 345.761,A -85,B 0,C 180,E1 -12897.769,E2 -12897.769} C_VEL
LIN {X 0,Y 361.373,Z 352.803,A -85,B 0,C 180,E1 -12899.732,E2 -12899.732} C_VEL
LIN {X 0,Y 360.917,Z 358.137,A -85,B 0,C 180,E1 -12901.72,E2 -12901.72} C_VEL
LIN {X 0,Y 360.52,Z 362.049,A -85,B 0,C 180,E1 -12903.751,E2 -12903.751} C_VEL
LIN {X 0,Y 360.276,Z 364.559,A -85,B 0,C 180,E1 -12905.819,E2 -12905.819} C_VEL
LIN {X 0,Y 360.201,Z 365.434,A -85,B 0,C 180,E1 -12907.219,E2 -12907.219} C_VEL
LIN {X 0,Y 360.199,Z 365.692,A -85,B 0,C 180,E1 -12908.699,E2 -12908.699} C_VEL
LIN {X 0,Y 360.329,Z 365.072,A -85,B 0,C 180,E1 -12910.478,E2 -12910.478} C_VEL
LIN {X 0,Y 360.58,Z 363.479,A -85,B 0,C 180,E1 -12912.214,E2 -12912.214} C_VEL
LIN {X 0,Y 360.881,Z 360.972,A -85,B 0,C 180,E1 -12913.9,E2 -12913.9} C_VEL
LIN {X 0,Y 361.416,Z 356.382,A -85,B 0,C 180,E1 -12916.014,E2 -12916.014} C_VEL
LIN {X 0,Y 362.146,Z 350.98,A -85,B 0,C 180,E1 -12917.842,E2 -12917.842} C_VEL
LIN {X 0,Y 363.005,Z 343.796,A -85,B 0,C 180,E1 -12919.712,E2 -12919.712} C_VEL
LIN {X 0,Y 363.943,Z 336.304,A -85,B 0,C 180,E1 -12921.267,E2 -12921.267} C_VEL
LIN {X 0,Y 365.078,Z 326.903,A -85,B 0,C 180,E1 -12922.845,E2 -12922.845} C_VEL
LIN {X 0,Y 366.182,Z 316.994,A -85,B 0,C 180,E1 -12924.171,E2 -12924.171} C_VEL
LIN {X 0,Y 367.36,Z 305.98,A -85,B 0,C 180,E1 -12925.351,E2 -12925.351} C_VEL
LIN {X 0,Y 368.329,Z 294.539,A -85,B 0,C 180,E1 -12926.322,E2 -12926.322} C_VEL
LIN {X 0,Y 369.156,Z 281.665,A -85,B 0,C 180,E1 -12927.142,E2 -12927.142} C_VEL
LIN {X 0,Y 369.744,Z 268.489,A -85,B 0,C 180,E1 -12927.736,E2 -12927.736} C_VEL
LIN {X 0,Y 370.188,Z 253.842,A -85,B 0,C 180,E1 -12928.124,E2 -12928.124} C_VEL
LIN {X 0,Y 371.908,Z 179.874,A -85,B 0,C 180,E1 -12929.668,E2 -12929.668} C_VEL
LIN {X 0,Y 369.908,Z 171.288,A -85,B 0,C 180,E1 -12930.009,E2 -12930.009} C_VEL
LIN {X 0,Y 363.589,Z 155.877,A -85,B 0,C 180,E1 -12930.875,E2 -12930.875} C_VEL
LIN {X 0,Y 361.946,Z 148.404,A -85,B 0,C 180,E1 -12933.028,E2 -12933.028} C_VEL
LIN {X 0,Y 361.908,Z 148.408,A -85,B 0,C 180,E1 -12935.934,E2 -12935.934} C_VEL
LIN {X 0,Y 361.89,Z 148.409,A -85,B 0,C 180,E1 -12939.54,E2 -12939.54} C_VEL
LIN {X 0,Y 361.932,Z 148.403,A -85,B 0,C 180,E1 -12943.067,E2 -12943.067} C_VEL
LIN {X 0,Y 362.003,Z 148.395,A -85,B 0,C 180,E1 -12946.529,E2 -12946.529} C_VEL
LIN {X 0,Y 362.004,Z 148.391,A -85,B 0,C 180,E1 -12949.938,E2 -12949.938} C_VEL
LIN {X 0,Y 362.127,Z 148.378,A -85,B 0,C 180,E1 -12953.314,E2 -12953.314} C_VEL
LIN {X 0,Y 362.269,Z 148.36,A -85,B 0,C 180,E1 -12957.777,E2 -12957.777} C_VEL
LIN {X 0,Y 362.18,Z 148.369,A -85,B 0,C 180,E1 -12961.112,E2 -12961.112} C_VEL
LIN {X 0,Y 362.262,Z 148.355,A -85,B 0,C 180,E1 -12962.224,E2 -12962.224} C_VEL
LIN {X 0,Y 362.128,Z 148.366,A -85,B 0,C 180,E1 -12966.688,E2 -12966.688} C_VEL
LIN {X 0,Y 361.998,Z 148.387,A -85,B 0,C 180,E1 -12970.064,E2 -12970.064} C_VEL
LIN {X 0,Y 361.956,Z 148.395,A -85,B 0,C 180,E1 -12973.868,E2 -12973.868} C_VEL
LIN {X 0,Y 361.88,Z 148.404,A -85,B 0,C 180,E1 -12978.104,E2 -12978.104} C_VEL
LIN {X 0,Y 361.824,Z 148.416,A -85,B 0,C 180,E1 -12981.658,E2 -12981.658} C_VEL
LIN {X 0,Y 361.856,Z 148.411,A -85,B 0,C 180,E1 -12985.296,E2 -12985.296} C_VEL
LIN {X 0,Y 361.861,Z 148.409,A -85,B 0,C 180,E1 -12989.074,E2 -12989.074} C_VEL
LIN {X 0,Y 361.851,Z 148.411,A -85,B 0,C 180,E1 -12992.945,E2 -12992.945} C_VEL
LIN {X 0,Y 361.872,Z 148.406,A -85,B 0,C 180,E1 -12995.637,E2 -12995.637} C_VEL
LIN {X 0,Y 361.831,Z 148.413,A -85,B 0,C 180,E1 -12999.018,E2 -12999.018} C_VEL
LIN {X 0,Y 361.837,Z 148.416,A -85,B 0,C 180,E1 -13002.829,E2 -13002.829} C_VEL
LIN {X 0,Y 361.821,Z 148.418,A -85,B 0,C 180,E1 -13005.947,E2 -13005.947} C_VEL
LIN {X 0,Y 361.817,Z 148.418,A -85,B 0,C 180,E1 -13009.249,E2 -13009.249} C_VEL
LIN {X 0,Y 361.869,Z 148.41,A -85,B 0,C 180,E1 -13012.981,E2 -13012.981} C_VEL
LIN {X 0,Y 361.864,Z 148.415,A -85,B 0,C 180,E1 -13016.63,E2 -13016.63} C_VEL
LIN {X 0,Y 361.864,Z 148.447,A -85,B 0,C 180,E1 -13018.711,E2 -13018.711} C_VEL
LIN {X 0,Y 364.377,Z 159.051,A -85,B 0,C 180,E1 -13021.486,E2 -13021.486} C_VEL
LIN {X 0,Y 366.256,Z 168.397,A -85,B 0,C 180,E1 -13023.81,E2 -13023.81} C_VEL
LIN {X 0,Y 366.223,Z 171.776,A -85,B 0,C 180,E1 -13024.576,E2 -13024.576} C_VEL
